(* PLC project marvel_thermovac, Institute of Astronomy Onto 0.0.1 *)
(* stored: creationDateTime 2025-01-01T00:00:00.0, modificationDateTime 2025-01-01T00:00:00.0 *)

{attribute 'qualified_only'}
TYPE TempControlStates : (idle := 0, warming_up := 1, active := 2);
END_TYPE

{attribute 'qualified_only'}
TYPE TempControlStatus : (unknown := 0, invalid_model := 1, idle := 2, warming_up := 3, active := 4) BYTE;
END_TYPE

TYPE OuterRoomParts : STRUCT
  {attribute 'TcHmiSymbol.Show'}
  tFloorE : TempMeasurement;  (* Floor sensor East *)
  {attribute 'TcHmiSymbol.Show'}
  tFloorW : TempMeasurement;  (* Floor sensor West *)
  {attribute 'TcHmiSymbol.Show'}
  tTopN : TempMeasurement;  (* Top sensor North *)
  {attribute 'TcHmiSymbol.Show'}
  tTopS : TempMeasurement;  (* Top sensor South *)
  {attribute 'TcHmiSymbol.Show'}
  ref : RefSensor;  (* Reference 'sensor' for calibration purposes *)
END_STRUCT;
END_TYPE

TYPE InnerRoomParts : STRUCT
  {attribute 'TcHmiSymbol.Show'}
  tAbove : TempMeasurement;  (* 1st temp sensor *)
  {attribute 'TcHmiSymbol.Show'}
  tBelow : TempMeasurement;  (* 2nd temp sensor *)
  {attribute 'TcHmiSymbol.Show'}
  tEast : TempMeasurement;  (* 3rd temp sensor *)
  {attribute 'TcHmiSymbol.Show'}
  tWest : TempMeasurement;  (* 4th temp sensor *)
  {attribute 'TcHmiSymbol.Show'}
  htDucts : Heater;  (* Test heater *)
  {attribute 'TcHmiSymbol.Show'}
  ref : RefSensor;  (* Reference 'sensor' for calibration purposes *)
END_STRUCT;
END_TYPE

TYPE VesselParts : STRUCT
  {attribute 'TcHmiSymbol.Show'}
  tLegNE : TempMeasurement;  (* Leg NE *)
  {attribute 'TcHmiSymbol.Show'}
  tLegNW : TempMeasurement;  (* Leg NW *)
  {attribute 'TcHmiSymbol.Show'}
  tLegSE : TempMeasurement;  (* Leg SE *)
  {attribute 'TcHmiSymbol.Show'}
  tLegSW : TempMeasurement;  (* Leg SW *)
  {attribute 'TcHmiSymbol.Show'}
  tLegTopNE : TempMeasurement;  (* Leg Top NE *)
  {attribute 'TcHmiSymbol.Show'}
  tLegTopNW : TempMeasurement;  (* Leg Top NW *)
  {attribute 'TcHmiSymbol.Show'}
  tLegTopSE : TempMeasurement;  (* Leg Top SE *)
  {attribute 'TcHmiSymbol.Show'}
  tLegTopSW : TempMeasurement;  (* Leg Top SW *)
  {attribute 'TcHmiSymbol.Show'}
  tBotNE : TempMeasurement;  (* Vessel Bottom NE *)
  {attribute 'TcHmiSymbol.Show'}
  tBotNW : TempMeasurement;  (* Vessel Bottom NW *)
  {attribute 'TcHmiSymbol.Show'}
  tBotSE : TempMeasurement;  (* Vessel Bottom SE *)
  {attribute 'TcHmiSymbol.Show'}
  tBotSW : TempMeasurement;  (* Vessel Bottom SW *)
  {attribute 'TcHmiSymbol.Show'}
  tCenter : TempMeasurement;  (* Centre *)
  {attribute 'TcHmiSymbol.Show'}
  tCenterTH10K : TempMeasurement;  (* Centre TH10K *)
  {attribute 'TcHmiSymbol.Show'}
  tSideN : TempMeasurement;  (* Vessel Side N *)
  {attribute 'TcHmiSymbol.Show'}
  tSideS : TempMeasurement;  (* Vessel Side S *)
  {attribute 'TcHmiSymbol.Show'}
  tSideE : TempMeasurement;  (* Vessel Side E *)
  {attribute 'TcHmiSymbol.Show'}
  tSideW : TempMeasurement;  (* Vessel Side W *)
  {attribute 'TcHmiSymbol.Show'}
  tLidN : TempMeasurement;  (* Vessel Lid N *)
  {attribute 'TcHmiSymbol.Show'}
  tLidS : TempMeasurement;  (* Vessel Lid S *)
  {attribute 'TcHmiSymbol.Show'}
  htLegNE : Heater;  (* Heater control for Leg NE *)
  {attribute 'TcHmiSymbol.Show'}
  htLegNW : Heater;  (* Heater control for Leg NW *)
  {attribute 'TcHmiSymbol.Show'}
  htLegSE : Heater;  (* Heater control for Leg SE *)
  {attribute 'TcHmiSymbol.Show'}
  htLegSW : Heater;  (* Heater control for Leg SW *)
  {attribute 'TcHmiSymbol.Show'}
  htLegTopNE : Heater;  (* Heater control for Leg Top NE *)
  {attribute 'TcHmiSymbol.Show'}
  htLegTopNW : Heater;  (* Heater control for Leg Top NW *)
  {attribute 'TcHmiSymbol.Show'}
  htLegTopSE : Heater;  (* Heater control for Leg Top SE *)
  {attribute 'TcHmiSymbol.Show'}
  htLegTopSW : Heater;  (* Heater control for Leg Top SW *)
  {attribute 'TcHmiSymbol.Show'}
  htBotNE : Heater;  (* Heater control for Vessel Bottom NE *)
  {attribute 'TcHmiSymbol.Show'}
  htBotNW : Heater;  (* Heater control for Vessel Bottom NW *)
  {attribute 'TcHmiSymbol.Show'}
  htBotSE : Heater;  (* Heater control for Vessel Bottom SE *)
  {attribute 'TcHmiSymbol.Show'}
  htBotSW : Heater;  (* Heater control for Vessel Bottom SW *)
  {attribute 'TcHmiSymbol.Show'}
  htSideN : Heater;  (* Heater control for Vessel Side NE *)
  {attribute 'TcHmiSymbol.Show'}
  htSideS : Heater;  (* Heater control for Vessel Side NW *)
  {attribute 'TcHmiSymbol.Show'}
  htSideE : Heater;  (* Heater control for Vessel Side SE *)
  {attribute 'TcHmiSymbol.Show'}
  htSideW : Heater;  (* Heater control for Vessel Side SW *)
  {attribute 'TcHmiSymbol.Show'}
  htLidN : Heater;  (* Heater control for Vessel Lid N *)
  {attribute 'TcHmiSymbol.Show'}
  htLidS : Heater;  (* Heater control for Vessel Lid S *)
  {attribute 'TcHmiSymbol.Show'}
  ref : RefSensor;  (* Reference 'sensor' for calibration purposes *)
END_STRUCT;
END_TYPE

TYPE ShieldParts : STRUCT
  {attribute 'TcHmiSymbol.Show'}
  tTopNE : TempMeasurement;  (* Shield top NE *)
  {attribute 'TcHmiSymbol.Show'}
  tTopNW : TempMeasurement;  (* Shield top NW *)
  {attribute 'TcHmiSymbol.Show'}
  tTopSE : TempMeasurement;  (* Shield top SE *)
  {attribute 'TcHmiSymbol.Show'}
  tTopSW : TempMeasurement;  (* Shield top SW *)
  {attribute 'TcHmiSymbol.Show'}
  tSideN : TempMeasurement;  (* Shield side N *)
  {attribute 'TcHmiSymbol.Show'}
  tSideS : TempMeasurement;  (* Shield side S *)
  {attribute 'TcHmiSymbol.Show'}
  tSideNE : TempMeasurement;  (* Shield side NE *)
  {attribute 'TcHmiSymbol.Show'}
  tSideSE : TempMeasurement;  (* Shield side SE *)
  {attribute 'TcHmiSymbol.Show'}
  tSideNW : TempMeasurement;  (* Shield side NW *)
  {attribute 'TcHmiSymbol.Show'}
  tSideSW : TempMeasurement;  (* Shield side SW *)
  {attribute 'TcHmiSymbol.Show'}
  tBotNE : TempMeasurement;  (* Shield bottom NE *)
  {attribute 'TcHmiSymbol.Show'}
  tBotNW : TempMeasurement;  (* Shield bottom NW *)
  {attribute 'TcHmiSymbol.Show'}
  tBotS : TempMeasurement;  (* Shield bottom S *)
  {attribute 'TcHmiSymbol.Show'}
  tCentre : TempMeasurement;  (* Shield centre *)
  {attribute 'TcHmiSymbol.Show'}
  tCentreTh10k : TempMeasurement;  (* Shield centre TH10k *)
  {attribute 'TcHmiSymbol.Show'}
  htTopNE : Heater;  (* Heater control for shield top NE *)
  {attribute 'TcHmiSymbol.Show'}
  htTopNW : Heater;  (* Heater control for shield top NW *)
  {attribute 'TcHmiSymbol.Show'}
  htTopSE : Heater;  (* Heater control for shield top SE *)
  {attribute 'TcHmiSymbol.Show'}
  htTopSW : Heater;  (* Heater control for shield top SW *)
  {attribute 'TcHmiSymbol.Show'}
  htSideN : Heater;  (* Heater control for shield side N *)
  {attribute 'TcHmiSymbol.Show'}
  htSideS : Heater;  (* Heater control for shield side S *)
  {attribute 'TcHmiSymbol.Show'}
  htSideNE : Heater;  (* Heater control for shield side NE *)
  {attribute 'TcHmiSymbol.Show'}
  htSideSE : Heater;  (* Heater control for shield side SE *)
  {attribute 'TcHmiSymbol.Show'}
  htSideNW : Heater;  (* Heater control for shield side NW *)
  {attribute 'TcHmiSymbol.Show'}
  htSideSW : Heater;  (* Heater control for shield side SW *)
  {attribute 'TcHmiSymbol.Show'}
  htBotNE : Heater;  (* Heater control for shield bottom NE *)
  {attribute 'TcHmiSymbol.Show'}
  htBotNW : Heater;  (* Heater control for shield bottom NW *)
  {attribute 'TcHmiSymbol.Show'}
  htBotS : Heater;  (* Heater control for shield bottom S *)
  {attribute 'TcHmiSymbol.Show'}
  htCentre : Heater;  (* Heater control for shield centre *)
  {attribute 'TcHmiSymbol.Show'}
  ref : RefSensor;  (* Reference 'sensor' for calibration purposes *)
END_STRUCT;
END_TYPE

TYPE BenchParts : STRUCT
  {attribute 'TcHmiSymbol.Show'}
  tCentre : TempMeasurement;  (* Bench centre *)
  {attribute 'TcHmiSymbol.Show'}
  tCentreTH10k : TempMeasurement;  (* Bench centre TH10k *)
  {attribute 'TcHmiSymbol.Show'}
  tCollBench : TempMeasurement;  (* Collimator bench *)
  {attribute 'TcHmiSymbol.Show'}
  tEchelleCryo : TempMeasurement;  (* Echelle cryo *)
  {attribute 'TcHmiSymbol.Show'}
  tCamCryo : TempMeasurement;  (* Camera cryo *)
  {attribute 'TcHmiSymbol.Show'}
  tColl : TempMeasurement;  (* Collimator *)
  {attribute 'TcHmiSymbol.Show'}
  tPrism : TempMeasurement;  (* Prism *)
  {attribute 'TcHmiSymbol.Show'}
  tEchelle : TempMeasurement;  (* Echelle *)
  {attribute 'TcHmiSymbol.Show'}
  tCam : TempMeasurement;  (* Camera *)
  {attribute 'TcHmiSymbol.Show'}
  tInOptics : TempMeasurement;  (* In-optics *)
  {attribute 'TcHmiSymbol.Show'}
  htCollBench : Heater;  (* Heater control for collimator bench *)
  {attribute 'TcHmiSymbol.Show'}
  htEchelleCryo : Heater;  (* Heater control for echelle cryo *)
  {attribute 'TcHmiSymbol.Show'}
  htCamCryo : Heater;  (* Heater control for camera cryo *)
  {attribute 'TcHmiSymbol.Show'}
  htEchellePrism : Heater;  (* Heater control for echelle/prism *)
  {attribute 'TcHmiSymbol.Show'}
  ref : RefSensor;  (* Reference 'sensor' for calibration purposes *)
END_STRUCT;
END_TYPE

TYPE CryoParts : STRUCT
  {attribute 'TcHmiSymbol.Show'}
  tRearOut : TempMeasurement;  (* Cryo rear outside *)
  {attribute 'TcHmiSymbol.Show'}
  tRearIn : TempMeasurement;  (* Cryo rear inside *)
  {attribute 'TcHmiSymbol.Show'}
  tFront : TempMeasurement;  (* Cryo front *)
  {attribute 'TcHmiSymbol.Show'}
  htRearOut : Heater;  (* Heater control for cryo rear outside *)
  {attribute 'TcHmiSymbol.Show'}
  htRearIn : Heater;  (* Heater control for cryo rear inside *)
  {attribute 'TcHmiSymbol.Show'}
  htRearFront : Heater;  (* Heater control for cryo front *)
  {attribute 'TcHmiSymbol.Show'}
  ref : RefSensor;  (* Reference 'sensor' for calibration purposes *)
END_STRUCT;
END_TYPE

TYPE ThermoParts : STRUCT
  {attribute 'TcHmiSymbol.Show'}
  outerRoom : OuterRoom;  (* State machine for the outer room temperature control *)
  {attribute 'TcHmiSymbol.Show'}
  innerRoom : InnerRoom;  (* State machine for the inner room temperature control *)
  {attribute 'TcHmiSymbol.Show'}
  vessel : Vessel;  (* State machine for the vessel temperature control *)
  {attribute 'TcHmiSymbol.Show'}
  shield : Shield;  (* State machine for the shield temperature control *)
  {attribute 'TcHmiSymbol.Show'}
  bench : Bench;  (* State machine for the bench temperature control *)
  {attribute 'TcHmiSymbol.Show'}
  cryo : Cryo;  (* State machine for the cryo temperature control *)
END_STRUCT;
END_TYPE

TYPE ThermoVacParts : STRUCT
  {attribute 'TcHmiSymbol.Show'}
  thermo : Thermo;  (* statemachine of the thermal control system *)
  {attribute 'TcHmiSymbol.Show'}
  vac : Vac;  (* statemachine of the vac control system *)
  {attribute 'TcHmiSymbol.Show'}
  configManager : ConfigManager;  (* The config manager (to load/save/activate configuration data) *)
END_STRUCT;
END_TYPE

TYPE TempMeasurementProcesses : STRUCT
  {attribute 'TcHmiSymbol.Show'}
  initialize : Process;  (* Initialize measurement *)
  {attribute 'TcHmiSymbol.Show'}
  clearPtp : Process;  (* Clear PTP values *)
END_STRUCT;
END_TYPE

TYPE HeaterProcesses : STRUCT
  {attribute 'TcHmiSymbol.Show'}
  initialize : Process;  (* Initialize the heater control *)
  {attribute 'TcHmiSymbol.Show'}
  reset : Process;  (* Reset the heater *)
  {attribute 'TcHmiSymbol.Show'}
  force : ForceHeater;  (* Force a certain power output to the heater *)
END_STRUCT;
END_TYPE

TYPE OuterRoomProcesses : STRUCT
  {attribute 'TcHmiSymbol.Show'}
  initialize : Process;  (* Start initializing *)
  {attribute 'TcHmiSymbol.Show'}
  start : Process;  (* Start warming up *)
  {attribute 'TcHmiSymbol.Show'}
  stop : Process;  (* Stop heating *)
  {attribute 'TcHmiSymbol.Show'}
  reset : Process;  (* Reset complete *)
  {attribute 'TcHmiSymbol.Show'}
  clearPtp : Process;  (* Clear the ptp values *)
  {attribute 'TcHmiSymbol.Show'}
  lock : Process;  (* Lock the outerroom control *)
  {attribute 'TcHmiSymbol.Show'}
  unlock : Process;  (* Unlock the outerroom control *)
END_STRUCT;
END_TYPE

TYPE InnerRoomProcesses : STRUCT
  {attribute 'TcHmiSymbol.Show'}
  initialize : Process;  (* Start initializing *)
  {attribute 'TcHmiSymbol.Show'}
  start : Process;  (* Start warming up *)
  {attribute 'TcHmiSymbol.Show'}
  stop : Process;  (* Stop heating *)
  {attribute 'TcHmiSymbol.Show'}
  reset : Process;  (* Reset complete *)
  {attribute 'TcHmiSymbol.Show'}
  clearPtp : Process;  (* Clear the ptp values *)
  {attribute 'TcHmiSymbol.Show'}
  lock : Process;  (* Lock the vessel control (e.g. when the vessel is opened) *)
  {attribute 'TcHmiSymbol.Show'}
  unlock : Process;  (* Unlock the vessel control (e.g. when the vessel is closed) *)
END_STRUCT;
END_TYPE

TYPE VesselProcesses : STRUCT
  {attribute 'TcHmiSymbol.Show'}
  initialize : Process;  (* Start initializing *)
  {attribute 'TcHmiSymbol.Show'}
  start : Process;  (* Start warming up *)
  {attribute 'TcHmiSymbol.Show'}
  stop : Process;  (* Stop heating *)
  {attribute 'TcHmiSymbol.Show'}
  reset : Process;  (* Reset complete *)
  {attribute 'TcHmiSymbol.Show'}
  clearPtp : Process;  (* Clear the ptp values *)
  {attribute 'TcHmiSymbol.Show'}
  lock : Process;  (* Lock the vessel control (e.g. when the vessel is opened) *)
  {attribute 'TcHmiSymbol.Show'}
  unlock : Process;  (* Unlock the vessel control (e.g. when the vessel is closed) *)
END_STRUCT;
END_TYPE

TYPE ShieldProcesses : STRUCT
  {attribute 'TcHmiSymbol.Show'}
  initialize : Process;  (* Start initializing *)
  {attribute 'TcHmiSymbol.Show'}
  start : Process;  (* Start warming up *)
  {attribute 'TcHmiSymbol.Show'}
  stop : Process;  (* Stop heating *)
  {attribute 'TcHmiSymbol.Show'}
  reset : Process;  (* Reset complete *)
  {attribute 'TcHmiSymbol.Show'}
  clearPtp : Process;  (* Clear the ptp values *)
  {attribute 'TcHmiSymbol.Show'}
  lock : Process;  (* Lock the shield control (e.g. when the shield is opened) *)
  {attribute 'TcHmiSymbol.Show'}
  unlock : Process;  (* Unlock the shield control (e.g. when the shield is closed) *)
END_STRUCT;
END_TYPE

TYPE BenchProcesses : STRUCT
  {attribute 'TcHmiSymbol.Show'}
  initialize : Process;  (* Start initializing *)
  {attribute 'TcHmiSymbol.Show'}
  start : Process;  (* Start warming up *)
  {attribute 'TcHmiSymbol.Show'}
  stop : Process;  (* Stop heating *)
  {attribute 'TcHmiSymbol.Show'}
  reset : Process;  (* Reset complete *)
  {attribute 'TcHmiSymbol.Show'}
  clearPtp : Process;  (* Clear the ptp values *)
  {attribute 'TcHmiSymbol.Show'}
  lock : Process;  (* Lock the bench control *)
  {attribute 'TcHmiSymbol.Show'}
  unlock : Process;  (* Unlock the bench control *)
END_STRUCT;
END_TYPE

TYPE CryoProcesses : STRUCT
  {attribute 'TcHmiSymbol.Show'}
  initialize : Process;  (* Start initializing *)
  {attribute 'TcHmiSymbol.Show'}
  start : Process;  (* Start warming up *)
  {attribute 'TcHmiSymbol.Show'}
  stop : Process;  (* Stop heating *)
  {attribute 'TcHmiSymbol.Show'}
  reset : Process;  (* Reset complete *)
  {attribute 'TcHmiSymbol.Show'}
  clearPtp : Process;  (* Clear the ptp values *)
  {attribute 'TcHmiSymbol.Show'}
  lock : Process;  (* Lock the cryo control *)
  {attribute 'TcHmiSymbol.Show'}
  unlock : Process;  (* Unlock the cryo control *)
END_STRUCT;
END_TYPE

TYPE ThermoProcesses : STRUCT
  {attribute 'TcHmiSymbol.Show'}
  initialize : Process;  (* Start initializing *)
  {attribute 'TcHmiSymbol.Show'}
  start : Process;  (* Start warming up *)
  {attribute 'TcHmiSymbol.Show'}
  stop : Process;  (* Stop heating *)
  {attribute 'TcHmiSymbol.Show'}
  clearPtp : Process;  (* Clear the ptp values *)
  {attribute 'TcHmiSymbol.Show'}
  reset : Process;  (* Reset complete *)
  {attribute 'TcHmiSymbol.Show'}
  lock : Process;  (* Lock the vessel control (e.g. when the vessel is opened) *)
  {attribute 'TcHmiSymbol.Show'}
  unlock : Process;  (* Unlock the vessel control (e.g. when the vessel is closed) *)
END_STRUCT;
END_TYPE

TYPE VacProcesses : STRUCT
  {attribute 'TcHmiSymbol.Show'}
  initialize : Process;  (* Start initializing *)
  {attribute 'TcHmiSymbol.Show'}
  reset : Process;  (* Reset complete *)
  {attribute 'TcHmiSymbol.Show'}
  lock : Process;  (* Lock the vessel control (e.g. when the vessel is opened) *)
  {attribute 'TcHmiSymbol.Show'}
  unlock : Process;  (* Unlock the vessel control (e.g. when the vessel is closed) *)
END_STRUCT;
END_TYPE

TYPE ThermoVacProcesses : STRUCT
  {attribute 'TcHmiSymbol.Show'}
  initialize : Process;  (* Start initializing *)
  {attribute 'TcHmiSymbol.Show'}
  reset : Process;  (* Reset complete *)
  {attribute 'TcHmiSymbol.Show'}
  lock : Process;  (* Lock the vessel control (e.g. when the vessel is opened) *)
  {attribute 'TcHmiSymbol.Show'}
  unlock : Process;  (* Unlock the vessel control (e.g. when the vessel is closed) *)
END_STRUCT;
END_TYPE

TYPE TempMeasurementStatuses : STRUCT
  {attribute 'OPC.UA.DA' := '1'}
  {attribute 'OPC.UA.DA.Access' := '1'}
  {attribute 'TcHmiSymbol.Show'}
  init : InitializationStatus;
  {attribute 'OPC.UA.DA' := '1'}
  {attribute 'OPC.UA.DA.Access' := '1'}
  {attribute 'TcHmiSymbol.Show'}
  enabled : EnabledStatus;  (* Is the measurement enabled? *)
  {attribute 'OPC.UA.DA' := '1'}
  {attribute 'OPC.UA.DA.Access' := '1'}
  {attribute 'TcHmiSymbol.Show'}
  health : HealthStatus;  (* Is the measurement OK? *)
  {attribute 'OPC.UA.DA' := '1'}
  {attribute 'OPC.UA.DA.Access' := '1'}
  {attribute 'TcHmiSymbol.Show'}
  alarm : HiHiLoLoAlarmStatus;  (* Alarm status *)
END_STRUCT;
END_TYPE

TYPE HeaterStatuses : STRUCT
  {attribute 'OPC.UA.DA' := '1'}
  {attribute 'OPC.UA.DA.Access' := '1'}
  {attribute 'TcHmiSymbol.Show'}
  init : InitializationStatus;
  {attribute 'OPC.UA.DA' := '1'}
  {attribute 'OPC.UA.DA.Access' := '1'}
  {attribute 'TcHmiSymbol.Show'}
  enabled : EnabledStatus;  (* Is the heater enabled? *)
  {attribute 'OPC.UA.DA' := '1'}
  {attribute 'OPC.UA.DA.Access' := '1'}
  {attribute 'TcHmiSymbol.Show'}
  health : HealthStatus;  (* Is the heater healthy? *)
  {attribute 'OPC.UA.DA' := '1'}
  {attribute 'OPC.UA.DA.Access' := '1'}
  {attribute 'TcHmiSymbol.Show'}
  alarm : HiHiLoLoAlarmStatus;  (* Alarm status *)
END_STRUCT;
END_TYPE

TYPE OuterRoomStatuses : STRUCT
  {attribute 'OPC.UA.DA' := '1'}
  {attribute 'OPC.UA.DA.Access' := '1'}
  {attribute 'TcHmiSymbol.Show'}
  init : InitializationStatus;
  {attribute 'OPC.UA.DA' := '1'}
  {attribute 'OPC.UA.DA.Access' := '1'}
  {attribute 'TcHmiSymbol.Show'}
  enabled : EnabledStatus;  (* Is the outer room enabled? *)
  {attribute 'OPC.UA.DA' := '1'}
  {attribute 'OPC.UA.DA.Access' := '1'}
  {attribute 'TcHmiSymbol.Show'}
  health : HealthStatus;  (* Is the outer room healthy? *)
  {attribute 'OPC.UA.DA' := '1'}
  {attribute 'OPC.UA.DA.Access' := '1'}
  {attribute 'TcHmiSymbol.Show'}
  control : TempControlStatus;  (* Actual state of the outer room *)
  {attribute 'OPC.UA.DA' := '1'}
  {attribute 'OPC.UA.DA.Access' := '1'}
  {attribute 'TcHmiSymbol.Show'}
  busy : BusyStatus;  (* Is the outer room busy with a procedure? *)
END_STRUCT;
END_TYPE

TYPE InnerRoomStatuses : STRUCT
  {attribute 'OPC.UA.DA' := '1'}
  {attribute 'OPC.UA.DA.Access' := '1'}
  {attribute 'TcHmiSymbol.Show'}
  init : InitializationStatus;
  {attribute 'OPC.UA.DA' := '1'}
  {attribute 'OPC.UA.DA.Access' := '1'}
  {attribute 'TcHmiSymbol.Show'}
  enabled : EnabledStatus;  (* Is the inner room enabled? *)
  {attribute 'OPC.UA.DA' := '1'}
  {attribute 'OPC.UA.DA.Access' := '1'}
  {attribute 'TcHmiSymbol.Show'}
  health : HealthStatus;  (* Is the vessel healthy? *)
  {attribute 'OPC.UA.DA' := '1'}
  {attribute 'OPC.UA.DA.Access' := '1'}
  {attribute 'TcHmiSymbol.Show'}
  control : TempControlStatus;  (* Actual state of the vessel *)
  {attribute 'OPC.UA.DA' := '1'}
  {attribute 'OPC.UA.DA.Access' := '1'}
  {attribute 'TcHmiSymbol.Show'}
  busy : BusyStatus;  (* Is the vessel busy with a procedure? *)
END_STRUCT;
END_TYPE

TYPE VesselStatuses : STRUCT
  {attribute 'OPC.UA.DA' := '1'}
  {attribute 'OPC.UA.DA.Access' := '1'}
  {attribute 'TcHmiSymbol.Show'}
  init : InitializationStatus;
  {attribute 'OPC.UA.DA' := '1'}
  {attribute 'OPC.UA.DA.Access' := '1'}
  {attribute 'TcHmiSymbol.Show'}
  enabled : EnabledStatus;  (* Is the vessel enabled? *)
  {attribute 'OPC.UA.DA' := '1'}
  {attribute 'OPC.UA.DA.Access' := '1'}
  {attribute 'TcHmiSymbol.Show'}
  health : HealthStatus;  (* Is the vessel healthy? *)
  {attribute 'OPC.UA.DA' := '1'}
  {attribute 'OPC.UA.DA.Access' := '1'}
  {attribute 'TcHmiSymbol.Show'}
  control : TempControlStatus;  (* Actual state of the vessel *)
  {attribute 'OPC.UA.DA' := '1'}
  {attribute 'OPC.UA.DA.Access' := '1'}
  {attribute 'TcHmiSymbol.Show'}
  busy : BusyStatus;  (* Is the vessel busy with a procedure? *)
END_STRUCT;
END_TYPE

TYPE ShieldStatuses : STRUCT
  {attribute 'OPC.UA.DA' := '1'}
  {attribute 'OPC.UA.DA.Access' := '1'}
  {attribute 'TcHmiSymbol.Show'}
  init : InitializationStatus;
  {attribute 'OPC.UA.DA' := '1'}
  {attribute 'OPC.UA.DA.Access' := '1'}
  {attribute 'TcHmiSymbol.Show'}
  enabled : EnabledStatus;  (* Is the shield enabled? *)
  {attribute 'OPC.UA.DA' := '1'}
  {attribute 'OPC.UA.DA.Access' := '1'}
  {attribute 'TcHmiSymbol.Show'}
  health : HealthStatus;  (* Is the shield healthy? *)
  {attribute 'OPC.UA.DA' := '1'}
  {attribute 'OPC.UA.DA.Access' := '1'}
  {attribute 'TcHmiSymbol.Show'}
  control : TempControlStatus;  (* Actual state of the shield *)
  {attribute 'OPC.UA.DA' := '1'}
  {attribute 'OPC.UA.DA.Access' := '1'}
  {attribute 'TcHmiSymbol.Show'}
  busy : BusyStatus;  (* Is the shield busy with a procedure? *)
END_STRUCT;
END_TYPE

TYPE BenchStatuses : STRUCT
  {attribute 'OPC.UA.DA' := '1'}
  {attribute 'OPC.UA.DA.Access' := '1'}
  {attribute 'TcHmiSymbol.Show'}
  init : InitializationStatus;
  {attribute 'OPC.UA.DA' := '1'}
  {attribute 'OPC.UA.DA.Access' := '1'}
  {attribute 'TcHmiSymbol.Show'}
  enabled : EnabledStatus;  (* Is the bench enabled? *)
  {attribute 'OPC.UA.DA' := '1'}
  {attribute 'OPC.UA.DA.Access' := '1'}
  {attribute 'TcHmiSymbol.Show'}
  health : HealthStatus;  (* Is the bench healthy? *)
  {attribute 'OPC.UA.DA' := '1'}
  {attribute 'OPC.UA.DA.Access' := '1'}
  {attribute 'TcHmiSymbol.Show'}
  control : TempControlStatus;  (* Actual state of the bench *)
  {attribute 'OPC.UA.DA' := '1'}
  {attribute 'OPC.UA.DA.Access' := '1'}
  {attribute 'TcHmiSymbol.Show'}
  busy : BusyStatus;  (* Is the bench busy with a procedure? *)
END_STRUCT;
END_TYPE

TYPE CryoStatuses : STRUCT
  {attribute 'OPC.UA.DA' := '1'}
  {attribute 'OPC.UA.DA.Access' := '1'}
  {attribute 'TcHmiSymbol.Show'}
  init : InitializationStatus;
  {attribute 'OPC.UA.DA' := '1'}
  {attribute 'OPC.UA.DA.Access' := '1'}
  {attribute 'TcHmiSymbol.Show'}
  enabled : EnabledStatus;  (* Is the cryo enabled? *)
  {attribute 'OPC.UA.DA' := '1'}
  {attribute 'OPC.UA.DA.Access' := '1'}
  {attribute 'TcHmiSymbol.Show'}
  health : HealthStatus;  (* Is the cryo healthy? *)
  {attribute 'OPC.UA.DA' := '1'}
  {attribute 'OPC.UA.DA.Access' := '1'}
  {attribute 'TcHmiSymbol.Show'}
  control : TempControlStatus;  (* Actual state of the cryo *)
  {attribute 'OPC.UA.DA' := '1'}
  {attribute 'OPC.UA.DA.Access' := '1'}
  {attribute 'TcHmiSymbol.Show'}
  busy : BusyStatus;  (* Is the cryo busy with a procedure? *)
END_STRUCT;
END_TYPE

TYPE ThermoStatuses : STRUCT
  {attribute 'OPC.UA.DA' := '1'}
  {attribute 'OPC.UA.DA.Access' := '1'}
  {attribute 'TcHmiSymbol.Show'}
  enabled : EnabledStatus;  (* Is the thermo control system enabled? *)
  {attribute 'OPC.UA.DA' := '1'}
  {attribute 'OPC.UA.DA.Access' := '1'}
  {attribute 'TcHmiSymbol.Show'}
  init : InitializationStatus;
  {attribute 'OPC.UA.DA' := '1'}
  {attribute 'OPC.UA.DA.Access' := '1'}
  {attribute 'TcHmiSymbol.Show'}
  health : HealthStatus;  (* Is the healthy? *)
  {attribute 'OPC.UA.DA' := '1'}
  {attribute 'OPC.UA.DA.Access' := '1'}
  {attribute 'TcHmiSymbol.Show'}
  busy : BusyStatus;  (* Is the vessel busy with a procedure? *)
  {attribute 'OPC.UA.DA' := '1'}
  {attribute 'OPC.UA.DA.Access' := '1'}
  {attribute 'TcHmiSymbol.Show'}
  control : TempControlStatus;  (* control state of the thermo control system *)
  {attribute 'OPC.UA.DA' := '1'}
  {attribute 'OPC.UA.DA.Access' := '1'}
  {attribute 'TcHmiSymbol.Show'}
  roomsStatHealth : HealthStatus;  (* Summerization of health states rooms, used for hmi *)
  {attribute 'OPC.UA.DA' := '1'}
  {attribute 'OPC.UA.DA.Access' := '1'}
  {attribute 'TcHmiSymbol.Show'}
  roomsStatBusy : BusyStatus;  (* Summerization of busy states rooms, used for hmi *)
END_STRUCT;
END_TYPE

TYPE VacStatuses : STRUCT
  {attribute 'OPC.UA.DA' := '1'}
  {attribute 'OPC.UA.DA.Access' := '1'}
  {attribute 'TcHmiSymbol.Show'}
  enabled : EnabledStatus;  (* Is the vac system enabled? *)
  {attribute 'OPC.UA.DA' := '1'}
  {attribute 'OPC.UA.DA.Access' := '1'}
  {attribute 'TcHmiSymbol.Show'}
  init : InitializationStatus;
  {attribute 'OPC.UA.DA' := '1'}
  {attribute 'OPC.UA.DA.Access' := '1'}
  {attribute 'TcHmiSymbol.Show'}
  health : HealthStatus;  (* Is the vessel healthy? *)
  {attribute 'OPC.UA.DA' := '1'}
  {attribute 'OPC.UA.DA.Access' := '1'}
  {attribute 'TcHmiSymbol.Show'}
  busy : BusyStatus;  (* Is the vessel busy with a procedure? *)
END_STRUCT;
END_TYPE

TYPE ThermoVacStatuses : STRUCT
  {attribute 'OPC.UA.DA' := '1'}
  {attribute 'OPC.UA.DA.Access' := '1'}
  {attribute 'TcHmiSymbol.Show'}
  init : InitializationStatus;
  {attribute 'OPC.UA.DA' := '1'}
  {attribute 'OPC.UA.DA.Access' := '1'}
  {attribute 'TcHmiSymbol.Show'}
  health : HealthStatus;  (* Is the vessel healthy? *)
  {attribute 'OPC.UA.DA' := '1'}
  {attribute 'OPC.UA.DA.Access' := '1'}
  {attribute 'TcHmiSymbol.Show'}
  busy : BusyStatus;  (* Is the vessel busy with a procedure? *)
END_STRUCT;
END_TYPE

TYPE HeaterConfig : STRUCT
  {attribute 'TcHmiSymbol.Show'}
  enabled : BOOL := TRUE;  (* True if the heater is enabled *)
  {attribute 'TcHmiSymbol.Show'}
  maxPower : LREAL := 100.0;  (* Maximum power of the heater *)
  {attribute 'TcHmiSymbol.Show'}
  Kp : LREAL;  (* proportional gain *)
  {attribute 'TcHmiSymbol.Show'}
  Tn : LREAL;  (* integral gain (in seconds) *)
  {attribute 'TcHmiSymbol.Show'}
  Tv : LREAL;  (* derivative gain D-T1 (in seconds) *)
  {attribute 'TcHmiSymbol.Show'}
  Td : LREAL;  (* derivative damping time D-T1 (in seconds) *)
END_STRUCT;
END_TYPE

TYPE MeasurementConfig2 : STRUCT
  {attribute 'TcHmiSymbol.Show'}
  enabled : BOOL := TRUE;  (* Is the quantity being measured? (Can be false e.g. if the sensor is deliberately not connected (yet).) *)
  {attribute 'TcHmiSymbol.Show'}
  gain : LREAL := 1.0;  (* Gain to be applied to the measured value (default: 1 = no gain) *)
  {attribute 'TcHmiSymbol.Show'}
  offset : LREAL;  (* Offset to be added to the measured value (default: 0 = no offset) *)
END_STRUCT;
END_TYPE

TYPE SimulationConfig : STRUCT
  {attribute 'TcHmiSymbol.Show'}
  ambient : LREAL;  (* starting temp of sensors *)
  {attribute 'TcHmiSymbol.Show'}
  heating : LREAL;  (* heating gain/factor (0-1) *)
  {attribute 'TcHmiSymbol.Show'}
  cooling : LREAL;  (* cooling factor (0-1) *)
  {attribute 'TcHmiSymbol.Show'}
  noise : LREAL;  (* factor (0-1) multiplied with random number (0-1) to create noise in the simulated temperature *)
END_STRUCT;
END_TYPE

TYPE SharedHeaterConfig : STRUCT
  {attribute 'TcHmiSymbol.Show'}
  simulation : SimulationConfig;
  {attribute 'TcHmiSymbol.Show'}
  hihilolo : HiHiLoLoAlarmConfig;  (* Alarm config for the heater's deviation from setpoint *)
  {attribute 'TcHmiSymbol.Show'}
  pwmPeriod : UINT := 1000;  (* period of the pwm signlas in ms *)
  {attribute 'TcHmiSymbol.Show'}
  pwmInstantUpdate : BOOL;  (* True if the PWM signal is updated instantly when the power changes *)
  {attribute 'TcHmiSymbol.Show'}
  maxPower : LREAL := 100.0;  (* Maximum total power of all heaters in percentage *)
  {attribute 'TcHmiSymbol.Show'}
  pidCycleTime : UINT := 100;  (* cycle time of the heater control loop in ms *)
  {attribute 'TcHmiSymbol.Show'}
  arwOnlyIpart : BOOL := TRUE;  (* True if the anti reset windup only applies to the integral part of the PID controller *)
END_STRUCT;
END_TYPE

TYPE SharedMeasurementConfig : STRUCT
  {attribute 'TcHmiSymbol.Show'}
  alarms : HiHiLoLoAlarmConfig;  (* Alarm config for the temperature sensors *)
  {attribute 'TcHmiSymbol.Show'}
  cycleTime : UINT := 100;  (* time in ms between temp measurements *)
  {attribute 'TcHmiSymbol.Show'}
  nrOfSamples : UINT := 50;  (* number of samples of the moving average *)
END_STRUCT;
END_TYPE

TYPE OuterRoomSharedConfig : STRUCT
  {attribute 'TcHmiSymbol.Show'}
  sensors : SharedMeasurementConfig;  (* Shared config for the temperature sensors *)
END_STRUCT;
END_TYPE

TYPE InnerRoomSharedConfig : STRUCT
  {attribute 'TcHmiSymbol.Show'}
  sensors : SharedMeasurementConfig;  (* Shared config for the temperature sensors *)
  {attribute 'TcHmiSymbol.Show'}
  heaters : SharedHeaterConfig;  (* Shared config for the heaters *)
END_STRUCT;
END_TYPE

TYPE VesselSharedConfig : STRUCT
  {attribute 'TcHmiSymbol.Show'}
  sensors : SharedMeasurementConfig;  (* Shared config for the temperature sensors in the vessel *)
  {attribute 'TcHmiSymbol.Show'}
  heaters : SharedHeaterConfig;  (* Shared config for the heaters in the vessel *)
END_STRUCT;
END_TYPE

TYPE ShieldSharedConfig : STRUCT
  {attribute 'TcHmiSymbol.Show'}
  sensors : SharedMeasurementConfig;  (* Shared config for the temperature sensors in the shield *)
  {attribute 'TcHmiSymbol.Show'}
  heaters : SharedHeaterConfig;  (* Shared config for the heaters in the shield *)
END_STRUCT;
END_TYPE

TYPE BenchSharedConfig : STRUCT
  {attribute 'TcHmiSymbol.Show'}
  sensors : SharedMeasurementConfig;  (* Shared config for the temperature sensors in the bench *)
  {attribute 'TcHmiSymbol.Show'}
  heaters : SharedHeaterConfig;  (* Shared config for the heaters in the bench *)
END_STRUCT;
END_TYPE

TYPE CryoSharedConfig : STRUCT
  {attribute 'TcHmiSymbol.Show'}
  sensors : SharedMeasurementConfig;  (* Shared config for the temperature sensors in the cryo *)
  {attribute 'TcHmiSymbol.Show'}
  heaters : SharedHeaterConfig;  (* Shared config for the heaters in the cryo *)
END_STRUCT;
END_TYPE

TYPE ThermoSharedConfig : STRUCT
  {attribute 'TcHmiSymbol.Show'}
  placeHolder : BOOL;  (* placeholder for the shared config of the thermo system, can be extended in the future *)
END_STRUCT;
END_TYPE

TYPE OuterRoomConfig : STRUCT
  {attribute 'TcHmiSymbol.Show'}
  enabled : BOOL := TRUE;  (* True if the outer room is enabled *)
  {attribute 'TcHmiSymbol.Show'}
  shared : OuterRoomSharedConfig;  (* Shared config for the outer room *)
  {attribute 'TcHmiSymbol.Show'}
  tFloorE : MeasurementConfig2;  (* Config for floor sensor East *)
  {attribute 'TcHmiSymbol.Show'}
  tFloorW : MeasurementConfig2;  (* Config for floor sensor West *)
  {attribute 'TcHmiSymbol.Show'}
  tTopN : MeasurementConfig2;  (* Config for top sensor North *)
  {attribute 'TcHmiSymbol.Show'}
  tTopS : MeasurementConfig2;  (* Config for top sensor South *)
END_STRUCT;
END_TYPE

TYPE InnerRoomConfig : STRUCT
  {attribute 'TcHmiSymbol.Show'}
  enabled : BOOL := TRUE;  (* True if the inner room is enabled *)
  {attribute 'TcHmiSymbol.Show'}
  shared : InnerRoomSharedConfig;  (* Config shared by inner room's parts *)
  {attribute 'TcHmiSymbol.Show'}
  isSimulated : BOOL;  (* True if the innerroom temperature control is in simulation mode *)
  {attribute 'TcHmiSymbol.Show'}
  setPointTarget : LREAL;  (* set point temperature in celsius *)
  {attribute 'TcHmiSymbol.Show'}
  rampVPos : LREAL;  (* velocity of temperature change in C/s while ramping up *)
  {attribute 'TcHmiSymbol.Show'}
  rampVNeg : LREAL;  (* velocity of temperature change in C/s while ramping down *)
  {attribute 'TcHmiSymbol.Show'}
  rampStart : LREAL;  (* temperature in celsius at which the ramp starts *)
  {attribute 'TcHmiSymbol.Show'}
  hihiPtp : LREAL;  (* Ptp value at which an alarm is given *)
  {attribute 'TcHmiSymbol.Show'}
  hiPtp : LREAL;  (* Ptp value at which a warning is given *)
  {attribute 'TcHmiSymbol.Show'}
  maxInitTime : LREAL := 120.0;  (* Maximum time in seconds before initialization is failed *)
  {attribute 'TcHmiSymbol.Show'}
  minSenRequired : INT := 4;  (* minimum number of sensors required to stay in operation *)
  {attribute 'TcHmiSymbol.Show'}
  tAbove : MeasurementConfig2;  (* Config for temp sensor above the vessel *)
  {attribute 'TcHmiSymbol.Show'}
  tBelow : MeasurementConfig2;  (* Config for temp sensor below the vessel *)
  {attribute 'TcHmiSymbol.Show'}
  tEast : MeasurementConfig2;  (* Config for temp sensor East of the vessel *)
  {attribute 'TcHmiSymbol.Show'}
  tWest : MeasurementConfig2;  (* Config for temp sensor West of the vessel *)
  {attribute 'TcHmiSymbol.Show'}
  htDucts : HeaterConfig;  (* Config for test heater *)
END_STRUCT;
END_TYPE

TYPE VesselConfig : STRUCT
  {attribute 'TcHmiSymbol.Show'}
  enabled : BOOL := TRUE;  (* True if the vessel is enabled *)
  {attribute 'TcHmiSymbol.Show'}
  shared : InnerRoomSharedConfig;  (* Config shared by vessels's parts *)
  {attribute 'TcHmiSymbol.Show'}
  isSimulated : BOOL;  (* True if the vessel temperature control is in simulation mode *)
  {attribute 'TcHmiSymbol.Show'}
  setPointTarget : LREAL;  (* set point temperature in celsius *)
  {attribute 'TcHmiSymbol.Show'}
  rampVPos : LREAL;  (* velocity of temperature change in C/s while ramping up *)
  {attribute 'TcHmiSymbol.Show'}
  rampVNeg : LREAL;  (* velocity of temperature change in C/s while ramping down *)
  {attribute 'TcHmiSymbol.Show'}
  rampStart : LREAL;  (* temperature in celsius at which the ramp starts *)
  {attribute 'TcHmiSymbol.Show'}
  hihiPtp : LREAL;  (* Ptp value at which an alarm is given *)
  {attribute 'TcHmiSymbol.Show'}
  hiPtp : LREAL;  (* Ptp value at which a warning is given *)
  {attribute 'TcHmiSymbol.Show'}
  maxInitTime : LREAL := 120.0;  (* Maximum time in seconds before initialization is failed *)
  {attribute 'TcHmiSymbol.Show'}
  tLegNE : MeasurementConfig2;  (* Config for Leg NE *)
  {attribute 'TcHmiSymbol.Show'}
  tLegNW : MeasurementConfig2;  (* Config for Leg NW *)
  {attribute 'TcHmiSymbol.Show'}
  tLegSE : MeasurementConfig2;  (* Config for Leg SE *)
  {attribute 'TcHmiSymbol.Show'}
  tLegSW : MeasurementConfig2;  (* Config for Leg SW *)
  {attribute 'TcHmiSymbol.Show'}
  tLegTopNE : MeasurementConfig2;  (* Config for Leg Top NE *)
  {attribute 'TcHmiSymbol.Show'}
  tLegTopNW : MeasurementConfig2;  (* Config for Leg Top NW *)
  {attribute 'TcHmiSymbol.Show'}
  tLegTopSE : MeasurementConfig2;  (* Config for Leg Top SE *)
  {attribute 'TcHmiSymbol.Show'}
  tLegTopSW : MeasurementConfig2;  (* Config for Leg Top SW *)
  {attribute 'TcHmiSymbol.Show'}
  tBotNE : MeasurementConfig2;  (* Config for Vessel Bottom NE *)
  {attribute 'TcHmiSymbol.Show'}
  tBotNW : MeasurementConfig2;  (* Config for Vessel Bottom NW *)
  {attribute 'TcHmiSymbol.Show'}
  tBotSE : MeasurementConfig2;  (* Config for Vessel Bottom SE *)
  {attribute 'TcHmiSymbol.Show'}
  tBotSW : MeasurementConfig2;  (* Config for Vessel Bottom SW *)
  {attribute 'TcHmiSymbol.Show'}
  tCenter : MeasurementConfig2;  (* Config for Centre *)
  {attribute 'TcHmiSymbol.Show'}
  tCenterTH10K : MeasurementConfig2;  (* Config for Centre TH10K *)
  {attribute 'TcHmiSymbol.Show'}
  tSideN : MeasurementConfig2;  (* Config for Vessel Side N *)
  {attribute 'TcHmiSymbol.Show'}
  tSideS : MeasurementConfig2;  (* Config for Vessel Side S *)
  {attribute 'TcHmiSymbol.Show'}
  tSideE : MeasurementConfig2;  (* Config for Vessel Side E *)
  {attribute 'TcHmiSymbol.Show'}
  tSideW : MeasurementConfig2;  (* Config for Vessel Side W *)
  {attribute 'TcHmiSymbol.Show'}
  tLidN : MeasurementConfig2;  (* Config for Vessel Lid N *)
  {attribute 'TcHmiSymbol.Show'}
  tLidS : MeasurementConfig2;  (* Config for Vessel Lid S *)
  {attribute 'TcHmiSymbol.Show'}
  htLegNE : HeaterConfig;  (* Config for heater Leg NE *)
  {attribute 'TcHmiSymbol.Show'}
  htLegNW : HeaterConfig;  (* Config for heater Leg NW *)
  {attribute 'TcHmiSymbol.Show'}
  htLegSE : HeaterConfig;  (* Config for heater Leg SE *)
  {attribute 'TcHmiSymbol.Show'}
  htLegSW : HeaterConfig;  (* Config for heater Leg SW *)
  {attribute 'TcHmiSymbol.Show'}
  htLegTopNE : HeaterConfig;  (* Config for heater Leg Top NE *)
  {attribute 'TcHmiSymbol.Show'}
  htLegTopNW : HeaterConfig;  (* Config for heater Leg Top NW *)
  {attribute 'TcHmiSymbol.Show'}
  htLegTopSE : HeaterConfig;  (* Config for heater Leg Top SE *)
  {attribute 'TcHmiSymbol.Show'}
  htLegTopSW : HeaterConfig;  (* Config for heater Leg Top SW *)
  {attribute 'TcHmiSymbol.Show'}
  htBotNE : HeaterConfig;  (* Config for heater Vessel Bottom NE *)
  {attribute 'TcHmiSymbol.Show'}
  htBotNW : HeaterConfig;  (* Config for heater Vessel Bottom NW *)
  {attribute 'TcHmiSymbol.Show'}
  htBotSE : HeaterConfig;  (* Config for heater Vessel Bottom SE *)
  {attribute 'TcHmiSymbol.Show'}
  htBotSW : HeaterConfig;  (* Config for heater Vessel Bottom SW *)
  {attribute 'TcHmiSymbol.Show'}
  htSideN : HeaterConfig;  (* Config for heater Vessel Side NE *)
  {attribute 'TcHmiSymbol.Show'}
  htSideS : HeaterConfig;  (* Config for heater Vessel Side NW *)
  {attribute 'TcHmiSymbol.Show'}
  htSideE : HeaterConfig;  (* Config for heater Vessel Side SE *)
  {attribute 'TcHmiSymbol.Show'}
  htSideW : HeaterConfig;  (* Config for heater Vessel Side SW *)
  {attribute 'TcHmiSymbol.Show'}
  htLidN : HeaterConfig;  (* Config for heater Vessel Lid N *)
  {attribute 'TcHmiSymbol.Show'}
  htLidS : HeaterConfig;  (* Config for heater Vessel Lid S *)
END_STRUCT;
END_TYPE

TYPE ShieldConfig : STRUCT
  {attribute 'TcHmiSymbol.Show'}
  enabled : BOOL := TRUE;  (* True if the shield is enabled *)
  {attribute 'TcHmiSymbol.Show'}
  shared : InnerRoomSharedConfig;  (* Config shared by shield's parts *)
  {attribute 'TcHmiSymbol.Show'}
  isSimulated : BOOL;  (* True if the shield temperature control is in simulation mode *)
  {attribute 'TcHmiSymbol.Show'}
  setPointTarget : LREAL;  (* set point temperature in celsius *)
  {attribute 'TcHmiSymbol.Show'}
  rampVPos : LREAL;  (* velocity of temperature change in C/s while ramping up *)
  {attribute 'TcHmiSymbol.Show'}
  rampVNeg : LREAL;  (* velocity of temperature change in C/s while ramping down *)
  {attribute 'TcHmiSymbol.Show'}
  rampStart : LREAL;  (* temperature in celsius at which the ramp starts *)
  {attribute 'TcHmiSymbol.Show'}
  hihiPtp : LREAL;  (* Ptp value at which an alarm is given *)
  {attribute 'TcHmiSymbol.Show'}
  hiPtp : LREAL;  (* Ptp value at which a warning is given *)
  {attribute 'TcHmiSymbol.Show'}
  maxInitTime : LREAL := 120.0;  (* Maximum time in seconds before initialization is failed *)
  {attribute 'TcHmiSymbol.Show'}
  tTopNE : MeasurementConfig2;  (* Config for shield top NE *)
  {attribute 'TcHmiSymbol.Show'}
  tTopNW : MeasurementConfig2;  (* Config for shield top NW *)
  {attribute 'TcHmiSymbol.Show'}
  tTopSE : MeasurementConfig2;  (* Config for shield top SE *)
  {attribute 'TcHmiSymbol.Show'}
  tTopSW : MeasurementConfig2;  (* Config for shield top SW *)
  {attribute 'TcHmiSymbol.Show'}
  tSideN : MeasurementConfig2;  (* Config for shield side N *)
  {attribute 'TcHmiSymbol.Show'}
  tSideS : MeasurementConfig2;  (* Config for shield side S *)
  {attribute 'TcHmiSymbol.Show'}
  tSideNE : MeasurementConfig2;  (* Config for shield side NE *)
  {attribute 'TcHmiSymbol.Show'}
  tSideSE : MeasurementConfig2;  (* Config for shield side SE *)
  {attribute 'TcHmiSymbol.Show'}
  tSideNW : MeasurementConfig2;  (* Config for shield side NW *)
  {attribute 'TcHmiSymbol.Show'}
  tSideSW : MeasurementConfig2;  (* Config for shield side SW *)
  {attribute 'TcHmiSymbol.Show'}
  tBotNE : MeasurementConfig2;  (* Config for shield bottom NE *)
  {attribute 'TcHmiSymbol.Show'}
  tBotNW : MeasurementConfig2;  (* Config for shield bottom NW *)
  {attribute 'TcHmiSymbol.Show'}
  tBotS : MeasurementConfig2;  (* Config for shield bottom S *)
  {attribute 'TcHmiSymbol.Show'}
  tCentre : MeasurementConfig2;  (* Config for shield centre *)
  {attribute 'TcHmiSymbol.Show'}
  tCentreTh10k : MeasurementConfig2;  (* Config for shield centre TH10k *)
  {attribute 'TcHmiSymbol.Show'}
  htTopNE : HeaterConfig;  (* Config for heater shield top NE *)
  {attribute 'TcHmiSymbol.Show'}
  htTopNW : HeaterConfig;  (* Config for heater shield top NW *)
  {attribute 'TcHmiSymbol.Show'}
  htTopSE : HeaterConfig;  (* Config for heater shield top SE *)
  {attribute 'TcHmiSymbol.Show'}
  htTopSW : HeaterConfig;  (* Config for heater shield top SW *)
  {attribute 'TcHmiSymbol.Show'}
  htSideN : HeaterConfig;  (* Config for heater shield side N *)
  {attribute 'TcHmiSymbol.Show'}
  htSideS : HeaterConfig;  (* Config for heater shield side S *)
  {attribute 'TcHmiSymbol.Show'}
  htSideNE : HeaterConfig;  (* Config for heater shield side NE *)
  {attribute 'TcHmiSymbol.Show'}
  htSideSE : HeaterConfig;  (* Config for heater shield side SE *)
  {attribute 'TcHmiSymbol.Show'}
  htSideNW : HeaterConfig;  (* Config for heater shield side NW *)
  {attribute 'TcHmiSymbol.Show'}
  htSideSW : HeaterConfig;  (* Config for heater shield side SW *)
  {attribute 'TcHmiSymbol.Show'}
  htBotNE : HeaterConfig;  (* Config for heater shield bottom NE *)
  {attribute 'TcHmiSymbol.Show'}
  htBotNW : HeaterConfig;  (* Config for heater shield bottom NW *)
  {attribute 'TcHmiSymbol.Show'}
  htBotS : HeaterConfig;  (* Config for heater shield bottom S *)
  {attribute 'TcHmiSymbol.Show'}
  htCentre : HeaterConfig;  (* Config for heater shield centre *)
END_STRUCT;
END_TYPE

TYPE BenchConfig : STRUCT
  {attribute 'TcHmiSymbol.Show'}
  enabled : BOOL := TRUE;  (* True if bench enabled *)
  {attribute 'TcHmiSymbol.Show'}
  shared : BenchSharedConfig;  (* Bench shared config *)
  {attribute 'TcHmiSymbol.Show'}
  tCentre : MeasurementConfig2;  (* Config for bench centre *)
  {attribute 'TcHmiSymbol.Show'}
  tCentreTH10k : MeasurementConfig2;  (* Bench centre TH10k sensor *)
  {attribute 'TcHmiSymbol.Show'}
  tCollBench : MeasurementConfig2;  (* Config for collimator bench *)
  {attribute 'TcHmiSymbol.Show'}
  tEchelleCryo : MeasurementConfig2;  (* Config for echelle cryo *)
  {attribute 'TcHmiSymbol.Show'}
  tCamCryo : MeasurementConfig2;  (* Config for camera cryo *)
  {attribute 'TcHmiSymbol.Show'}
  tColl : MeasurementConfig2;  (* Config for collimator *)
  {attribute 'TcHmiSymbol.Show'}
  tPrism : MeasurementConfig2;  (* Config for prism *)
  {attribute 'TcHmiSymbol.Show'}
  tEchelle : MeasurementConfig2;  (* Config for echelle *)
  {attribute 'TcHmiSymbol.Show'}
  tCam : MeasurementConfig2;  (* Config for camera *)
  {attribute 'TcHmiSymbol.Show'}
  tInOptics : MeasurementConfig2;  (* Config for in-optics *)
  {attribute 'TcHmiSymbol.Show'}
  htCollBench : HeaterConfig;  (* Config for heater collimator bench *)
  {attribute 'TcHmiSymbol.Show'}
  htEchelleCryo : HeaterConfig;  (* Config for heater echelle cryo *)
  {attribute 'TcHmiSymbol.Show'}
  htCamCryo : HeaterConfig;  (* Config for heater camera cryo *)
  {attribute 'TcHmiSymbol.Show'}
  htEchellePrism : HeaterConfig;  (* Config for heater echelle/prism *)
END_STRUCT;
END_TYPE

TYPE CryoConfig : STRUCT
  {attribute 'TcHmiSymbol.Show'}
  enabled : BOOL := TRUE;  (* True if cryo enabled *)
  {attribute 'TcHmiSymbol.Show'}
  shared : CryoSharedConfig;  (* Cryo shared config *)
  {attribute 'TcHmiSymbol.Show'}
  tRearOut : MeasurementConfig2;  (* Cryo rear outside sensor *)
  {attribute 'TcHmiSymbol.Show'}
  tRearIn : MeasurementConfig2;  (* Cryo rear inside sensor *)
  {attribute 'TcHmiSymbol.Show'}
  tFront : MeasurementConfig2;  (* Cryo front sensor *)
  {attribute 'TcHmiSymbol.Show'}
  htRearOut : HeaterConfig;  (* Heater cryo rear outside *)
  {attribute 'TcHmiSymbol.Show'}
  htRearIn : HeaterConfig;  (* Heater cryo rear inside *)
  {attribute 'TcHmiSymbol.Show'}
  htRearFront : HeaterConfig;  (* Heater cryo front *)
END_STRUCT;
END_TYPE

TYPE ThermoConfig : STRUCT
  {attribute 'TcHmiSymbol.Show'}
  enabled : BOOL := TRUE;  (* True if thermo enabled *)
  {attribute 'TcHmiSymbol.Show'}
  outerRoom : OuterRoomConfig;  (* Config for the outer room *)
  {attribute 'TcHmiSymbol.Show'}
  innerRoom : InnerRoomConfig;  (* Config for the inner room *)
  {attribute 'TcHmiSymbol.Show'}
  vessel : VesselConfig;  (* Config for the vessel *)
  {attribute 'TcHmiSymbol.Show'}
  shield : ShieldConfig;  (* Config for the shield *)
  {attribute 'TcHmiSymbol.Show'}
  bench : BenchConfig;  (* Config for the bench *)
  {attribute 'TcHmiSymbol.Show'}
  cryo : CryoConfig;  (* Config for the cryo *)
  {attribute 'TcHmiSymbol.Show'}
  shared : ThermoSharedConfig;  (* Shared config for the thermo system *)
END_STRUCT;
END_TYPE

TYPE VacConfig : STRUCT
  {attribute 'TcHmiSymbol.Show'}
  enabled : BOOL;  (* True if the vac system is enabled *)
END_STRUCT;
END_TYPE

TYPE ThermoVacConfig : STRUCT
  {attribute 'TcHmiSymbol.Show'}
  thermo : ThermoConfig;  (* Thermo config *)
  {attribute 'TcHmiSymbol.Show'}
  vac : VacConfig;  (* Vacuum config *)
END_STRUCT;
END_TYPE

TYPE ForceHeaterArgs : STRUCT
  {attribute 'TcHmiSymbol.Show'}
  power : REAL;
END_STRUCT;
END_TYPE

TYPE M_SM_RefSensor : STRUCT
  {attribute 'OPC.UA.DA' := '1'}
  {attribute 'OPC.UA.DA.Access' := '1'}
  {attribute 'TcHmiSymbol.Show'}
  actualStatus : STRING;
  {attribute 'OPC.UA.DA' := '1'}
  {attribute 'OPC.UA.DA.Access' := '1'}
  {attribute 'TcHmiSymbol.Show'}
  value : LREAL;
END_STRUCT;
END_TYPE

TYPE M_SM_TempMeasurement : STRUCT
  {attribute 'OPC.UA.DA' := '1'}
  {attribute 'OPC.UA.DA.Access' := '1'}
  {attribute 'TcHmiSymbol.Show'}
  isSimulated : BOOL;
  {attribute 'OPC.UA.DA' := '1'}
  {attribute 'OPC.UA.DA.Access' := '1'}
  {attribute 'TcHmiSymbol.Show'}
  actualStatus : STRING;
  {attribute 'OPC.UA.DA' := '1'}
  {attribute 'OPC.UA.DA.Access' := '1'}
  {attribute 'TcHmiSymbol.Show'}
  value : LREAL;
  {attribute 'OPC.UA.DA' := '1'}
  {attribute 'OPC.UA.DA.Access' := '1'}
  {attribute 'TcHmiSymbol.Show'}
  ptp1 : LREAL;
  {attribute 'OPC.UA.DA' := '1'}
  {attribute 'OPC.UA.DA.Access' := '1'}
  {attribute 'TcHmiSymbol.Show'}
  ptp2 : LREAL;
  {attribute 'OPC.UA.DA' := '1'}
  {attribute 'TcHmiSymbol.Show'}
  stat : TempMeasurementStatuses;
  {attribute 'OPC.UA.DA' := '1'}
  {attribute 'TcHmiSymbol.Show'}
  proc : M_SM_TempMeasurementProcesses;
END_STRUCT;
END_TYPE

TYPE M_SM_Heater : STRUCT
  {attribute 'OPC.UA.DA' := '1'}
  {attribute 'OPC.UA.DA.Access' := '1'}
  {attribute 'TcHmiSymbol.Show'}
  setPoint : LREAL;
  {attribute 'OPC.UA.DA' := '1'}
  {attribute 'OPC.UA.DA.Access' := '1'}
  {attribute 'TcHmiSymbol.Show'}
  temp : LREAL;
  {attribute 'OPC.UA.DA' := '1'}
  {attribute 'OPC.UA.DA.Access' := '1'}
  {attribute 'TcHmiSymbol.Show'}
  isSimulated : BOOL;
  {attribute 'OPC.UA.DA' := '1'}
  {attribute 'OPC.UA.DA.Access' := '1'}
  {attribute 'TcHmiSymbol.Show'}
  actualStatus : STRING;
  {attribute 'OPC.UA.DA' := '1'}
  {attribute 'OPC.UA.DA.Access' := '1'}
  {attribute 'TcHmiSymbol.Show'}
  power : LREAL;
  {attribute 'OPC.UA.DA' := '1'}
  {attribute 'OPC.UA.DA.Access' := '1'}
  {attribute 'TcHmiSymbol.Show'}
  deviation : LREAL;
  {attribute 'OPC.UA.DA' := '1'}
  {attribute 'OPC.UA.DA.Access' := '1'}
  {attribute 'TcHmiSymbol.Show'}
  isForced : BOOL;
  {attribute 'OPC.UA.DA' := '1'}
  {attribute 'OPC.UA.DA.Access' := '1'}
  {attribute 'TcHmiSymbol.Show'}
  simTemp : LREAL;
  {attribute 'OPC.UA.DA' := '1'}
  {attribute 'TcHmiSymbol.Show'}
  stat : HeaterStatuses;
  {attribute 'OPC.UA.DA' := '1'}
  {attribute 'TcHmiSymbol.Show'}
  proc : M_SM_HeaterProcesses;
END_STRUCT;
END_TYPE

TYPE M_SM_OuterRoom : STRUCT
  {attribute 'OPC.UA.DA' := '1'}
  {attribute 'OPC.UA.DA.Access' := '1'}
  {attribute 'TcHmiSymbol.Show'}
  actualStatus : STRING;
  {attribute 'OPC.UA.DA' := '1'}
  {attribute 'TcHmiSymbol.Show'}
  stat : OuterRoomStatuses;
  {attribute 'OPC.UA.DA' := '1'}
  {attribute 'TcHmiSymbol.Show'}
  parts : M_SM_OuterRoomParts;
  {attribute 'OPC.UA.DA' := '1'}
  {attribute 'TcHmiSymbol.Show'}
  proc : M_SM_OuterRoomProcesses;
END_STRUCT;
END_TYPE

TYPE M_SM_InnerRoom : STRUCT
  {attribute 'OPC.UA.DA' := '1'}
  {attribute 'OPC.UA.DA.Access' := '1'}
  {attribute 'TcHmiSymbol.Show'}
  actualStatus : STRING;
  {attribute 'OPC.UA.DA' := '1'}
  {attribute 'OPC.UA.DA.Access' := '1'}
  {attribute 'TcHmiSymbol.Show'}
  setPoint : LREAL;
  {attribute 'OPC.UA.DA' := '1'}
  {attribute 'OPC.UA.DA.Access' := '1'}
  {attribute 'TcHmiSymbol.Show'}
  avgTemp : LREAL;
  {attribute 'OPC.UA.DA' := '1'}
  {attribute 'OPC.UA.DA.Access' := '1'}
  {attribute 'TcHmiSymbol.Show'}
  avgPower : LREAL;
  {attribute 'OPC.UA.DA' := '1'}
  {attribute 'OPC.UA.DA.Access' := '1'}
  {attribute 'TcHmiSymbol.Show'}
  totalPower : LREAL;
  {attribute 'OPC.UA.DA' := '1'}
  {attribute 'OPC.UA.DA.Access' := '1'}
  {attribute 'TcHmiSymbol.Show'}
  ptpAvgTemp : ARRAY[1..5] OF LREAL;
  {attribute 'OPC.UA.DA' := '1'}
  {attribute 'OPC.UA.DA.Access' := '1'}
  {attribute 'TcHmiSymbol.Show'}
  ptpAllTemp : ARRAY[1..5] OF LREAL;
  {attribute 'OPC.UA.DA' := '1'}
  {attribute 'TcHmiSymbol.Show'}
  stat : InnerRoomStatuses;
  {attribute 'OPC.UA.DA' := '1'}
  {attribute 'TcHmiSymbol.Show'}
  parts : M_SM_InnerRoomParts;
  {attribute 'OPC.UA.DA' := '1'}
  {attribute 'TcHmiSymbol.Show'}
  proc : M_SM_InnerRoomProcesses;
END_STRUCT;
END_TYPE

TYPE M_SM_Vessel : STRUCT
  {attribute 'OPC.UA.DA' := '1'}
  {attribute 'OPC.UA.DA.Access' := '1'}
  {attribute 'TcHmiSymbol.Show'}
  tStatBottomOk : BOOL;
  {attribute 'OPC.UA.DA' := '1'}
  {attribute 'OPC.UA.DA.Access' := '1'}
  {attribute 'TcHmiSymbol.Show'}
  tStatLidOk : BOOL;
  {attribute 'OPC.UA.DA' := '1'}
  {attribute 'OPC.UA.DA.Access' := '1'}
  {attribute 'TcHmiSymbol.Show'}
  actualStatus : STRING;
  {attribute 'OPC.UA.DA' := '1'}
  {attribute 'OPC.UA.DA.Access' := '1'}
  {attribute 'TcHmiSymbol.Show'}
  setPoint : LREAL;
  {attribute 'OPC.UA.DA' := '1'}
  {attribute 'OPC.UA.DA.Access' := '1'}
  {attribute 'TcHmiSymbol.Show'}
  avgTemp : LREAL;
  {attribute 'OPC.UA.DA' := '1'}
  {attribute 'OPC.UA.DA.Access' := '1'}
  {attribute 'TcHmiSymbol.Show'}
  avgPower : LREAL;
  {attribute 'OPC.UA.DA' := '1'}
  {attribute 'OPC.UA.DA.Access' := '1'}
  {attribute 'TcHmiSymbol.Show'}
  totalPower : LREAL;
  {attribute 'OPC.UA.DA' := '1'}
  {attribute 'OPC.UA.DA.Access' := '1'}
  {attribute 'TcHmiSymbol.Show'}
  ptpAvgTemp : ARRAY[1..5] OF LREAL;
  {attribute 'OPC.UA.DA' := '1'}
  {attribute 'OPC.UA.DA.Access' := '1'}
  {attribute 'TcHmiSymbol.Show'}
  ptpAllTemp : ARRAY[1..5] OF LREAL;
  {attribute 'OPC.UA.DA' := '1'}
  {attribute 'OPC.UA.DA.Access' := '1'}
  {attribute 'TcHmiSymbol.Show'}
  tStatBottomPwr : BOOL;
  {attribute 'OPC.UA.DA' := '1'}
  {attribute 'OPC.UA.DA.Access' := '1'}
  {attribute 'TcHmiSymbol.Show'}
  tStatLidPwr : BOOL;
  {attribute 'OPC.UA.DA' := '1'}
  {attribute 'TcHmiSymbol.Show'}
  stat : VesselStatuses;
  {attribute 'OPC.UA.DA' := '1'}
  {attribute 'TcHmiSymbol.Show'}
  parts : M_SM_VesselParts;
  {attribute 'OPC.UA.DA' := '1'}
  {attribute 'TcHmiSymbol.Show'}
  proc : M_SM_VesselProcesses;
END_STRUCT;
END_TYPE

TYPE M_SM_Shield : STRUCT
  {attribute 'OPC.UA.DA' := '1'}
  {attribute 'OPC.UA.DA.Access' := '1'}
  {attribute 'TcHmiSymbol.Show'}
  actualStatus : STRING;
  {attribute 'OPC.UA.DA' := '1'}
  {attribute 'OPC.UA.DA.Access' := '1'}
  {attribute 'TcHmiSymbol.Show'}
  setPoint : LREAL;
  {attribute 'OPC.UA.DA' := '1'}
  {attribute 'OPC.UA.DA.Access' := '1'}
  {attribute 'TcHmiSymbol.Show'}
  avgTemp : LREAL;
  {attribute 'OPC.UA.DA' := '1'}
  {attribute 'OPC.UA.DA.Access' := '1'}
  {attribute 'TcHmiSymbol.Show'}
  avgPower : LREAL;
  {attribute 'OPC.UA.DA' := '1'}
  {attribute 'OPC.UA.DA.Access' := '1'}
  {attribute 'TcHmiSymbol.Show'}
  totalPower : LREAL;
  {attribute 'OPC.UA.DA' := '1'}
  {attribute 'OPC.UA.DA.Access' := '1'}
  {attribute 'TcHmiSymbol.Show'}
  ptpAvgTemp : ARRAY[1..5] OF LREAL;
  {attribute 'OPC.UA.DA' := '1'}
  {attribute 'OPC.UA.DA.Access' := '1'}
  {attribute 'TcHmiSymbol.Show'}
  ptpAllTemp : ARRAY[1..5] OF LREAL;
  {attribute 'OPC.UA.DA' := '1'}
  {attribute 'TcHmiSymbol.Show'}
  stat : ShieldStatuses;
  {attribute 'OPC.UA.DA' := '1'}
  {attribute 'TcHmiSymbol.Show'}
  parts : M_SM_ShieldParts;
  {attribute 'OPC.UA.DA' := '1'}
  {attribute 'TcHmiSymbol.Show'}
  proc : M_SM_ShieldProcesses;
END_STRUCT;
END_TYPE

TYPE M_SM_Bench : STRUCT
  {attribute 'OPC.UA.DA' := '1'}
  {attribute 'OPC.UA.DA.Access' := '1'}
  {attribute 'TcHmiSymbol.Show'}
  actualStatus : STRING;
  {attribute 'OPC.UA.DA' := '1'}
  {attribute 'TcHmiSymbol.Show'}
  stat : BenchStatuses;
  {attribute 'OPC.UA.DA' := '1'}
  {attribute 'TcHmiSymbol.Show'}
  parts : M_SM_BenchParts;
  {attribute 'OPC.UA.DA' := '1'}
  {attribute 'TcHmiSymbol.Show'}
  proc : M_SM_BenchProcesses;
END_STRUCT;
END_TYPE

TYPE M_SM_Cryo : STRUCT
  {attribute 'OPC.UA.DA' := '1'}
  {attribute 'OPC.UA.DA.Access' := '1'}
  {attribute 'TcHmiSymbol.Show'}
  tStatCryoRearOk : BOOL;
  {attribute 'OPC.UA.DA' := '1'}
  {attribute 'OPC.UA.DA.Access' := '1'}
  {attribute 'TcHmiSymbol.Show'}
  actualStatus : STRING;
  {attribute 'OPC.UA.DA' := '1'}
  {attribute 'OPC.UA.DA.Access' := '1'}
  {attribute 'TcHmiSymbol.Show'}
  tStatCryoRearPwr : BOOL;
  {attribute 'OPC.UA.DA' := '1'}
  {attribute 'TcHmiSymbol.Show'}
  stat : CryoStatuses;
  {attribute 'OPC.UA.DA' := '1'}
  {attribute 'TcHmiSymbol.Show'}
  parts : M_SM_CryoParts;
  {attribute 'OPC.UA.DA' := '1'}
  {attribute 'TcHmiSymbol.Show'}
  proc : M_SM_CryoProcesses;
END_STRUCT;
END_TYPE

TYPE M_SM_Thermo : STRUCT
  {attribute 'OPC.UA.DA' := '1'}
  {attribute 'OPC.UA.DA.Access' := '1'}
  {attribute 'TcHmiSymbol.Show'}
  actualStatus : STRING;
  {attribute 'OPC.UA.DA' := '1'}
  {attribute 'TcHmiSymbol.Show'}
  stat : ThermoStatuses;
  {attribute 'OPC.UA.DA' := '1'}
  {attribute 'TcHmiSymbol.Show'}
  parts : M_SM_ThermoParts;
  {attribute 'OPC.UA.DA' := '1'}
  {attribute 'TcHmiSymbol.Show'}
  proc : M_SM_ThermoProcesses;
END_STRUCT;
END_TYPE

TYPE M_SM_Vac : STRUCT
  {attribute 'OPC.UA.DA' := '1'}
  {attribute 'OPC.UA.DA.Access' := '1'}
  {attribute 'TcHmiSymbol.Show'}
  actualStatus : STRING;
  {attribute 'OPC.UA.DA' := '1'}
  {attribute 'TcHmiSymbol.Show'}
  stat : VacStatuses;
  {attribute 'OPC.UA.DA' := '1'}
  {attribute 'TcHmiSymbol.Show'}
  proc : M_SM_VacProcesses;
END_STRUCT;
END_TYPE

TYPE M_SM_ThermoVac : STRUCT
  {attribute 'OPC.UA.DA' := '1'}
  {attribute 'OPC.UA.DA.Access' := '3'}
  {attribute 'TcHmiSymbol.Show'}
  editableConfig : ThermoVacConfig;
  {attribute 'OPC.UA.DA' := '1'}
  {attribute 'OPC.UA.DA.Access' := '1'}
  {attribute 'TcHmiSymbol.Show'}
  actualStatus : STRING;
  {attribute 'OPC.UA.DA' := '1'}
  {attribute 'OPC.UA.DA.Access' := '1'}
  {attribute 'TcHmiSymbol.Show'}
  config : ThermoVacConfig;
  {attribute 'OPC.UA.DA' := '1'}
  {attribute 'TcHmiSymbol.Show'}
  stat : ThermoVacStatuses;
  {attribute 'OPC.UA.DA' := '1'}
  {attribute 'TcHmiSymbol.Show'}
  parts : M_SM_ThermoVacParts;
  {attribute 'OPC.UA.DA' := '1'}
  {attribute 'TcHmiSymbol.Show'}
  proc : M_SM_ThermoVacProcesses;
END_STRUCT;
END_TYPE

TYPE M_ForceHeater : STRUCT
  {attribute 'OPC.UA.DA' := '1'}
  {attribute 'OPC.UA.DA.Access' := '3'}
  {attribute 'TcHmiSymbol.Show'}
  set : ForceHeaterArgs;
END_STRUCT;
END_TYPE

TYPE M_SM_TempMeasurementProcesses : STRUCT
  {attribute 'TcHmiSymbol.Show'}
  initialize : M_Process;
  {attribute 'TcHmiSymbol.Show'}
  clearPtp : M_Process;
END_STRUCT;
END_TYPE

TYPE M_SM_HeaterProcesses : STRUCT
  {attribute 'TcHmiSymbol.Show'}
  initialize : M_Process;
  {attribute 'TcHmiSymbol.Show'}
  reset : M_Process;
  {attribute 'TcHmiSymbol.Show'}
  force : M_ForceHeater;
END_STRUCT;
END_TYPE

TYPE M_SM_OuterRoomParts : STRUCT
  {attribute 'TcHmiSymbol.Show'}
  tFloorE : M_TempMeasurement;
  {attribute 'TcHmiSymbol.Show'}
  tFloorW : M_TempMeasurement;
  {attribute 'TcHmiSymbol.Show'}
  tTopN : M_TempMeasurement;
  {attribute 'TcHmiSymbol.Show'}
  tTopS : M_TempMeasurement;
  {attribute 'TcHmiSymbol.Show'}
  ref : M_RefSensor;
END_STRUCT;
END_TYPE

TYPE M_SM_OuterRoomProcesses : STRUCT
  {attribute 'TcHmiSymbol.Show'}
  initialize : M_Process;
  {attribute 'TcHmiSymbol.Show'}
  start : M_Process;
  {attribute 'TcHmiSymbol.Show'}
  stop : M_Process;
  {attribute 'TcHmiSymbol.Show'}
  reset : M_Process;
  {attribute 'TcHmiSymbol.Show'}
  clearPtp : M_Process;
  {attribute 'TcHmiSymbol.Show'}
  lock : M_Process;
  {attribute 'TcHmiSymbol.Show'}
  unlock : M_Process;
END_STRUCT;
END_TYPE

TYPE M_SM_InnerRoomParts : STRUCT
  {attribute 'TcHmiSymbol.Show'}
  tAbove : M_TempMeasurement;
  {attribute 'TcHmiSymbol.Show'}
  tBelow : M_TempMeasurement;
  {attribute 'TcHmiSymbol.Show'}
  tEast : M_TempMeasurement;
  {attribute 'TcHmiSymbol.Show'}
  tWest : M_TempMeasurement;
  {attribute 'TcHmiSymbol.Show'}
  htDucts : M_Heater;
  {attribute 'TcHmiSymbol.Show'}
  ref : M_RefSensor;
END_STRUCT;
END_TYPE

TYPE M_SM_InnerRoomProcesses : STRUCT
  {attribute 'TcHmiSymbol.Show'}
  initialize : M_Process;
  {attribute 'TcHmiSymbol.Show'}
  start : M_Process;
  {attribute 'TcHmiSymbol.Show'}
  stop : M_Process;
  {attribute 'TcHmiSymbol.Show'}
  reset : M_Process;
  {attribute 'TcHmiSymbol.Show'}
  clearPtp : M_Process;
  {attribute 'TcHmiSymbol.Show'}
  lock : M_Process;
  {attribute 'TcHmiSymbol.Show'}
  unlock : M_Process;
END_STRUCT;
END_TYPE

TYPE M_SM_VesselParts : STRUCT
  {attribute 'TcHmiSymbol.Show'}
  tLegNE : M_TempMeasurement;
  {attribute 'TcHmiSymbol.Show'}
  tLegNW : M_TempMeasurement;
  {attribute 'TcHmiSymbol.Show'}
  tLegSE : M_TempMeasurement;
  {attribute 'TcHmiSymbol.Show'}
  tLegSW : M_TempMeasurement;
  {attribute 'TcHmiSymbol.Show'}
  tLegTopNE : M_TempMeasurement;
  {attribute 'TcHmiSymbol.Show'}
  tLegTopNW : M_TempMeasurement;
  {attribute 'TcHmiSymbol.Show'}
  tLegTopSE : M_TempMeasurement;
  {attribute 'TcHmiSymbol.Show'}
  tLegTopSW : M_TempMeasurement;
  {attribute 'TcHmiSymbol.Show'}
  tBotNE : M_TempMeasurement;
  {attribute 'TcHmiSymbol.Show'}
  tBotNW : M_TempMeasurement;
  {attribute 'TcHmiSymbol.Show'}
  tBotSE : M_TempMeasurement;
  {attribute 'TcHmiSymbol.Show'}
  tBotSW : M_TempMeasurement;
  {attribute 'TcHmiSymbol.Show'}
  tCenter : M_TempMeasurement;
  {attribute 'TcHmiSymbol.Show'}
  tCenterTH10K : M_TempMeasurement;
  {attribute 'TcHmiSymbol.Show'}
  tSideN : M_TempMeasurement;
  {attribute 'TcHmiSymbol.Show'}
  tSideS : M_TempMeasurement;
  {attribute 'TcHmiSymbol.Show'}
  tSideE : M_TempMeasurement;
  {attribute 'TcHmiSymbol.Show'}
  tSideW : M_TempMeasurement;
  {attribute 'TcHmiSymbol.Show'}
  tLidN : M_TempMeasurement;
  {attribute 'TcHmiSymbol.Show'}
  tLidS : M_TempMeasurement;
  {attribute 'TcHmiSymbol.Show'}
  htLegNE : M_Heater;
  {attribute 'TcHmiSymbol.Show'}
  htLegNW : M_Heater;
  {attribute 'TcHmiSymbol.Show'}
  htLegSE : M_Heater;
  {attribute 'TcHmiSymbol.Show'}
  htLegSW : M_Heater;
  {attribute 'TcHmiSymbol.Show'}
  htLegTopNE : M_Heater;
  {attribute 'TcHmiSymbol.Show'}
  htLegTopNW : M_Heater;
  {attribute 'TcHmiSymbol.Show'}
  htLegTopSE : M_Heater;
  {attribute 'TcHmiSymbol.Show'}
  htLegTopSW : M_Heater;
  {attribute 'TcHmiSymbol.Show'}
  htBotNE : M_Heater;
  {attribute 'TcHmiSymbol.Show'}
  htBotNW : M_Heater;
  {attribute 'TcHmiSymbol.Show'}
  htBotSE : M_Heater;
  {attribute 'TcHmiSymbol.Show'}
  htBotSW : M_Heater;
  {attribute 'TcHmiSymbol.Show'}
  htSideN : M_Heater;
  {attribute 'TcHmiSymbol.Show'}
  htSideS : M_Heater;
  {attribute 'TcHmiSymbol.Show'}
  htSideE : M_Heater;
  {attribute 'TcHmiSymbol.Show'}
  htSideW : M_Heater;
  {attribute 'TcHmiSymbol.Show'}
  htLidN : M_Heater;
  {attribute 'TcHmiSymbol.Show'}
  htLidS : M_Heater;
  {attribute 'TcHmiSymbol.Show'}
  ref : M_RefSensor;
END_STRUCT;
END_TYPE

TYPE M_SM_VesselProcesses : STRUCT
  {attribute 'TcHmiSymbol.Show'}
  initialize : M_Process;
  {attribute 'TcHmiSymbol.Show'}
  start : M_Process;
  {attribute 'TcHmiSymbol.Show'}
  stop : M_Process;
  {attribute 'TcHmiSymbol.Show'}
  reset : M_Process;
  {attribute 'TcHmiSymbol.Show'}
  clearPtp : M_Process;
  {attribute 'TcHmiSymbol.Show'}
  lock : M_Process;
  {attribute 'TcHmiSymbol.Show'}
  unlock : M_Process;
END_STRUCT;
END_TYPE

TYPE M_SM_ShieldParts : STRUCT
  {attribute 'TcHmiSymbol.Show'}
  tTopNE : M_TempMeasurement;
  {attribute 'TcHmiSymbol.Show'}
  tTopNW : M_TempMeasurement;
  {attribute 'TcHmiSymbol.Show'}
  tTopSE : M_TempMeasurement;
  {attribute 'TcHmiSymbol.Show'}
  tTopSW : M_TempMeasurement;
  {attribute 'TcHmiSymbol.Show'}
  tSideN : M_TempMeasurement;
  {attribute 'TcHmiSymbol.Show'}
  tSideS : M_TempMeasurement;
  {attribute 'TcHmiSymbol.Show'}
  tSideNE : M_TempMeasurement;
  {attribute 'TcHmiSymbol.Show'}
  tSideSE : M_TempMeasurement;
  {attribute 'TcHmiSymbol.Show'}
  tSideNW : M_TempMeasurement;
  {attribute 'TcHmiSymbol.Show'}
  tSideSW : M_TempMeasurement;
  {attribute 'TcHmiSymbol.Show'}
  tBotNE : M_TempMeasurement;
  {attribute 'TcHmiSymbol.Show'}
  tBotNW : M_TempMeasurement;
  {attribute 'TcHmiSymbol.Show'}
  tBotS : M_TempMeasurement;
  {attribute 'TcHmiSymbol.Show'}
  tCentre : M_TempMeasurement;
  {attribute 'TcHmiSymbol.Show'}
  tCentreTh10k : M_TempMeasurement;
  {attribute 'TcHmiSymbol.Show'}
  htTopNE : M_Heater;
  {attribute 'TcHmiSymbol.Show'}
  htTopNW : M_Heater;
  {attribute 'TcHmiSymbol.Show'}
  htTopSE : M_Heater;
  {attribute 'TcHmiSymbol.Show'}
  htTopSW : M_Heater;
  {attribute 'TcHmiSymbol.Show'}
  htSideN : M_Heater;
  {attribute 'TcHmiSymbol.Show'}
  htSideS : M_Heater;
  {attribute 'TcHmiSymbol.Show'}
  htSideNE : M_Heater;
  {attribute 'TcHmiSymbol.Show'}
  htSideSE : M_Heater;
  {attribute 'TcHmiSymbol.Show'}
  htSideNW : M_Heater;
  {attribute 'TcHmiSymbol.Show'}
  htSideSW : M_Heater;
  {attribute 'TcHmiSymbol.Show'}
  htBotNE : M_Heater;
  {attribute 'TcHmiSymbol.Show'}
  htBotNW : M_Heater;
  {attribute 'TcHmiSymbol.Show'}
  htBotS : M_Heater;
  {attribute 'TcHmiSymbol.Show'}
  htCentre : M_Heater;
  {attribute 'TcHmiSymbol.Show'}
  ref : M_RefSensor;
END_STRUCT;
END_TYPE

TYPE M_SM_ShieldProcesses : STRUCT
  {attribute 'TcHmiSymbol.Show'}
  initialize : M_Process;
  {attribute 'TcHmiSymbol.Show'}
  start : M_Process;
  {attribute 'TcHmiSymbol.Show'}
  stop : M_Process;
  {attribute 'TcHmiSymbol.Show'}
  reset : M_Process;
  {attribute 'TcHmiSymbol.Show'}
  clearPtp : M_Process;
  {attribute 'TcHmiSymbol.Show'}
  lock : M_Process;
  {attribute 'TcHmiSymbol.Show'}
  unlock : M_Process;
END_STRUCT;
END_TYPE

TYPE M_SM_BenchParts : STRUCT
  {attribute 'TcHmiSymbol.Show'}
  tCentre : M_TempMeasurement;
  {attribute 'TcHmiSymbol.Show'}
  tCentreTH10k : M_TempMeasurement;
  {attribute 'TcHmiSymbol.Show'}
  tCollBench : M_TempMeasurement;
  {attribute 'TcHmiSymbol.Show'}
  tEchelleCryo : M_TempMeasurement;
  {attribute 'TcHmiSymbol.Show'}
  tCamCryo : M_TempMeasurement;
  {attribute 'TcHmiSymbol.Show'}
  tColl : M_TempMeasurement;
  {attribute 'TcHmiSymbol.Show'}
  tPrism : M_TempMeasurement;
  {attribute 'TcHmiSymbol.Show'}
  tEchelle : M_TempMeasurement;
  {attribute 'TcHmiSymbol.Show'}
  tCam : M_TempMeasurement;
  {attribute 'TcHmiSymbol.Show'}
  tInOptics : M_TempMeasurement;
  {attribute 'TcHmiSymbol.Show'}
  htCollBench : M_Heater;
  {attribute 'TcHmiSymbol.Show'}
  htEchelleCryo : M_Heater;
  {attribute 'TcHmiSymbol.Show'}
  htCamCryo : M_Heater;
  {attribute 'TcHmiSymbol.Show'}
  htEchellePrism : M_Heater;
  {attribute 'TcHmiSymbol.Show'}
  ref : M_RefSensor;
END_STRUCT;
END_TYPE

TYPE M_SM_BenchProcesses : STRUCT
  {attribute 'TcHmiSymbol.Show'}
  initialize : M_Process;
  {attribute 'TcHmiSymbol.Show'}
  start : M_Process;
  {attribute 'TcHmiSymbol.Show'}
  stop : M_Process;
  {attribute 'TcHmiSymbol.Show'}
  reset : M_Process;
  {attribute 'TcHmiSymbol.Show'}
  clearPtp : M_Process;
  {attribute 'TcHmiSymbol.Show'}
  lock : M_Process;
  {attribute 'TcHmiSymbol.Show'}
  unlock : M_Process;
END_STRUCT;
END_TYPE

TYPE M_SM_CryoParts : STRUCT
  {attribute 'TcHmiSymbol.Show'}
  tRearOut : M_TempMeasurement;
  {attribute 'TcHmiSymbol.Show'}
  tRearIn : M_TempMeasurement;
  {attribute 'TcHmiSymbol.Show'}
  tFront : M_TempMeasurement;
  {attribute 'TcHmiSymbol.Show'}
  htRearOut : M_Heater;
  {attribute 'TcHmiSymbol.Show'}
  htRearIn : M_Heater;
  {attribute 'TcHmiSymbol.Show'}
  htRearFront : M_Heater;
  {attribute 'TcHmiSymbol.Show'}
  ref : M_RefSensor;
END_STRUCT;
END_TYPE

TYPE M_SM_CryoProcesses : STRUCT
  {attribute 'TcHmiSymbol.Show'}
  initialize : M_Process;
  {attribute 'TcHmiSymbol.Show'}
  start : M_Process;
  {attribute 'TcHmiSymbol.Show'}
  stop : M_Process;
  {attribute 'TcHmiSymbol.Show'}
  reset : M_Process;
  {attribute 'TcHmiSymbol.Show'}
  clearPtp : M_Process;
  {attribute 'TcHmiSymbol.Show'}
  lock : M_Process;
  {attribute 'TcHmiSymbol.Show'}
  unlock : M_Process;
END_STRUCT;
END_TYPE

TYPE M_SM_ThermoParts : STRUCT
  {attribute 'TcHmiSymbol.Show'}
  outerRoom : M_OuterRoom;
  {attribute 'TcHmiSymbol.Show'}
  innerRoom : M_InnerRoom;
  {attribute 'TcHmiSymbol.Show'}
  vessel : M_Vessel;
  {attribute 'TcHmiSymbol.Show'}
  shield : M_Shield;
  {attribute 'TcHmiSymbol.Show'}
  bench : M_Bench;
  {attribute 'TcHmiSymbol.Show'}
  cryo : M_Cryo;
END_STRUCT;
END_TYPE

TYPE M_SM_ThermoProcesses : STRUCT
  {attribute 'TcHmiSymbol.Show'}
  initialize : M_Process;
  {attribute 'TcHmiSymbol.Show'}
  start : M_Process;
  {attribute 'TcHmiSymbol.Show'}
  stop : M_Process;
  {attribute 'TcHmiSymbol.Show'}
  clearPtp : M_Process;
  {attribute 'TcHmiSymbol.Show'}
  reset : M_Process;
  {attribute 'TcHmiSymbol.Show'}
  lock : M_Process;
  {attribute 'TcHmiSymbol.Show'}
  unlock : M_Process;
END_STRUCT;
END_TYPE

TYPE M_SM_VacProcesses : STRUCT
  {attribute 'TcHmiSymbol.Show'}
  initialize : M_Process;
  {attribute 'TcHmiSymbol.Show'}
  reset : M_Process;
  {attribute 'TcHmiSymbol.Show'}
  lock : M_Process;
  {attribute 'TcHmiSymbol.Show'}
  unlock : M_Process;
END_STRUCT;
END_TYPE

TYPE M_SM_ThermoVacParts : STRUCT
  {attribute 'TcHmiSymbol.Show'}
  thermo : M_Thermo;
  {attribute 'TcHmiSymbol.Show'}
  vac : M_Vac;
  {attribute 'TcHmiSymbol.Show'}
  configManager : M_ConfigManager;
END_STRUCT;
END_TYPE

TYPE M_SM_ThermoVacProcesses : STRUCT
  {attribute 'TcHmiSymbol.Show'}
  initialize : M_Process;
  {attribute 'TcHmiSymbol.Show'}
  reset : M_Process;
  {attribute 'TcHmiSymbol.Show'}
  lock : M_Process;
  {attribute 'TcHmiSymbol.Show'}
  unlock : M_Process;
END_STRUCT;
END_TYPE

{attribute 'TcRpcEnable' := '1'}
FUNCTION F_TempControlStatus : TempControlStatus
  VAR_INPUT
    superState : BOOL := TRUE;  (* Super state (TRUE if the super state is active, or if there is no super state) *)
    isActive : BOOL;  (* True if the temp control is active (not idle) *)
    isWarmingUp : BOOL;  (* True if the system warming up *)
  END_VAR

              IF NOT(superState) THEN
    F_TempControlStatus := TempControlStatus.unknown;
ELSIF (NOT(isActive)) AND (NOT(isWarmingUp)) THEN
    F_TempControlStatus := TempControlStatus.idle;
ELSIF isWarmingUp THEN
    F_TempControlStatus := TempControlStatus.warming_up;
ELSIF isActive AND (NOT(isWarmingUp)) THEN
    F_TempControlStatus := TempControlStatus.active;
ELSE
    F_TempControlStatus := TempControlStatus.invalid_model;
END_IF;

            
END_FUNCTION

FUNCTION_BLOCK SM_RefSensor
  VAR_OUTPUT
    {attribute 'OPC.UA.DA' := '1'}
    {attribute 'OPC.UA.DA.Access' := '1'}
    actualStatus : STRING(50);  (* Current status description *)
    {attribute 'OPC.UA.DA' := '1'}
    {attribute 'OPC.UA.DA.Access' := '1'}
    value : LREAL;  (* Measured value *)
  END_VAR

            
          

METHOD _copyFromModel_SM_RefSensor
  VAR_IN_OUT
    {attribute 'OPC.UA.DA' := '0'}
    model : M_SM_RefSensor;
  END_VAR
                  
                
END_METHOD

METHOD _copyToModel_SM_RefSensor
  VAR_IN_OUT
    {attribute 'OPC.UA.DA' := '0'}
    model : M_SM_RefSensor;
  END_VAR
                  model.actualStatus := THIS^.actualStatus;
model.value := THIS^.value;

                
END_METHOD
END_FUNCTION_BLOCK

FUNCTION_BLOCK SM_TempMeasurement
  VAR_INPUT
    {attribute 'OPC.UA.DA' := '1'}
    {attribute 'OPC.UA.DA.Access' := '1'}
    isSimulated : BOOL;
    {attribute 'OPC.UA.DA' := '0'}
    rawValue AT %I* : REAL;  (* Raw measured value *)
    {attribute 'OPC.UA.DA' := '0'}
    error : BOOL;  (* True if sensor error *)
  END_VAR
  VAR_OUTPUT
    {attribute 'OPC.UA.DA' := '1'}
    {attribute 'OPC.UA.DA.Access' := '1'}
    actualStatus : STRING(50);  (* Current status description *)
    {attribute 'OPC.UA.DA' := '1'}
    {attribute 'OPC.UA.DA.Access' := '1'}
    value : LREAL;  (* Measured value *)
    {attribute 'OPC.UA.DA' := '1'}
    {attribute 'OPC.UA.DA.Access' := '1'}
    ptp1 : LREAL;
    {attribute 'OPC.UA.DA' := '1'}
    {attribute 'OPC.UA.DA.Access' := '1'}
    ptp2 : LREAL;
    {attribute 'OPC.UA.DA' := '1'}
    stat : TempMeasurementStatuses;  (* Statuses of the state machine *)
    {attribute 'OPC.UA.DA' := '1'}
    proc : TempMeasurementProcesses;  (* Processes of the state machine *)
  END_VAR
  VAR_IN_OUT
    {attribute 'OPC.UA.DA' := '0'}
    config_ref : MeasurementConfig2;  (* Reference to the config *)
    {attribute 'OPC.UA.DA' := '0'}
    sharedConfig_ref : SharedMeasurementConfig;  (* Reference to sensor alarm config *)
  END_VAR

            stat.enabled := F_EnabledStatus(
    superState := TRUE,
    isEnabled := config_ref.enabled);
stat.health := F_HealthStatus(
    superState := stat.enabled = EnabledStatus.enabled,
    isGood := NOT((stat.alarm = HiHiLoLoAlarmStatus.hiHi) OR ((stat.alarm = HiHiLoLoAlarmStatus.loLo) OR error)),
    hasWarning := (stat.alarm = HiHiLoLoAlarmStatus.hi) OR ((stat.alarm = HiHiLoLoAlarmStatus.lo) OR (NOT(sharedConfig_ref.alarms.enabled))));
proc.initialize( isEnabled := NOT((stat.init = InitializationStatus.locked) OR (stat.enabled = EnabledStatus.disabled)) );
proc.clearPtp( isEnabled := stat.init = InitializationStatus.initialized );

          

METHOD _copyFromModel_SM_TempMeasurement
  VAR_IN_OUT
    {attribute 'OPC.UA.DA' := '0'}
    model : M_SM_TempMeasurement;
  END_VAR
                  THIS^.proc.initialize._copyFromModel_Process( model := model.proc.initialize );
THIS^.proc.clearPtp._copyFromModel_Process( model := model.proc.clearPtp );

                
END_METHOD

METHOD _copyToModel_SM_TempMeasurement
  VAR_IN_OUT
    {attribute 'OPC.UA.DA' := '0'}
    model : M_SM_TempMeasurement;
  END_VAR
                  model.isSimulated := THIS^.isSimulated;
model.actualStatus := THIS^.actualStatus;
model.value := THIS^.value;
model.ptp1 := THIS^.ptp1;
model.ptp2 := THIS^.ptp2;
model.stat := THIS^.stat;
THIS^.proc.initialize._copyToModel_Process( model := model.proc.initialize );
THIS^.proc.clearPtp._copyToModel_Process( model := model.proc.clearPtp );

                
END_METHOD
END_FUNCTION_BLOCK

FUNCTION_BLOCK SM_Heater
  VAR_INPUT
    {attribute 'OPC.UA.DA' := '1'}
    {attribute 'OPC.UA.DA.Access' := '1'}
    setPoint : LREAL;  (* Current set point of the heater in kelvin *)
    {attribute 'OPC.UA.DA' := '1'}
    {attribute 'OPC.UA.DA.Access' := '1'}
    temp : LREAL;  (* Associated temperature of the heater in kelvin *)
    {attribute 'OPC.UA.DA' := '1'}
    {attribute 'OPC.UA.DA.Access' := '1'}
    isSimulated : BOOL;
  END_VAR
  VAR_OUTPUT
    {attribute 'OPC.UA.DA' := '1'}
    {attribute 'OPC.UA.DA.Access' := '1'}
    actualStatus : STRING(50);  (* Current status description *)
    {attribute 'OPC.UA.DA' := '1'}
    {attribute 'OPC.UA.DA.Access' := '1'}
    power : LREAL;  (* Current power of the heater in percentage *)
    {attribute 'OPC.UA.DA' := '1'}
    {attribute 'OPC.UA.DA.Access' := '1'}
    deviation : LREAL;  (* Current error between set point and associated temperature *)
    {attribute 'OPC.UA.DA' := '1'}
    {attribute 'OPC.UA.DA.Access' := '1'}
    isForced : BOOL;  (* True if the heater power is forced (overwriting the normal control) *)
    {attribute 'OPC.UA.DA' := '1'}
    {attribute 'OPC.UA.DA.Access' := '1'}
    simTemp : LREAL;  (* Simulated temperature for testing the heater control *)
    {attribute 'OPC.UA.DA' := '1'}
    stat : HeaterStatuses;  (* Statuses of the state machine *)
    {attribute 'OPC.UA.DA' := '1'}
    proc : HeaterProcesses;  (* Processes of the state machine *)
  END_VAR
  VAR_IN_OUT
    {attribute 'OPC.UA.DA' := '0'}
    config_ref : HeaterConfig;  (* Reference to the heater config *)
    {attribute 'OPC.UA.DA' := '0'}
    sharedConfig_ref : SharedHeaterConfig;  (* Reference to the shared heater config *)
    {attribute 'OPC.UA.DA' := '0'}
    operator_ref : OperatorStatus;  (* Shared operator status *)
  END_VAR

            stat.enabled := F_EnabledStatus(
    superState := TRUE,
    isEnabled := config_ref.enabled);
proc.initialize( isEnabled := NOT((stat.init = InitializationStatus.locked) OR (stat.init = InitializationStatus.initializing)) );
proc.reset( isEnabled := TRUE );
proc.force( isEnabled := (operator_ref = OperatorStatus.tech) AND ((NOT(isForced)) AND ((stat.enabled = EnabledStatus.enabled) AND (stat.init = InitializationStatus.initialized))) );

          

METHOD _copyFromModel_SM_Heater
  VAR_IN_OUT
    {attribute 'OPC.UA.DA' := '0'}
    model : M_SM_Heater;
  END_VAR
                  THIS^.proc.initialize._copyFromModel_Process( model := model.proc.initialize );
THIS^.proc.reset._copyFromModel_Process( model := model.proc.reset );
THIS^.proc.force._copyFromModel_ForceHeater( model := model.proc.force );

                
END_METHOD

METHOD _copyToModel_SM_Heater
  VAR_IN_OUT
    {attribute 'OPC.UA.DA' := '0'}
    model : M_SM_Heater;
  END_VAR
                  model.setPoint := THIS^.setPoint;
model.temp := THIS^.temp;
model.isSimulated := THIS^.isSimulated;
model.actualStatus := THIS^.actualStatus;
model.power := THIS^.power;
model.deviation := THIS^.deviation;
model.isForced := THIS^.isForced;
model.simTemp := THIS^.simTemp;
model.stat := THIS^.stat;
THIS^.proc.initialize._copyToModel_Process( model := model.proc.initialize );
THIS^.proc.reset._copyToModel_Process( model := model.proc.reset );
THIS^.proc.force._copyToModel_ForceHeater( model := model.proc.force );

                
END_METHOD
END_FUNCTION_BLOCK

FUNCTION_BLOCK SM_OuterRoom
  VAR_OUTPUT
    {attribute 'OPC.UA.DA' := '1'}
    {attribute 'OPC.UA.DA.Access' := '1'}
    actualStatus : STRING(50);  (* Current status description *)
    {attribute 'OPC.UA.DA' := '1'}
    stat : OuterRoomStatuses;  (* Statuses of the state machine *)
    {attribute 'OPC.UA.DA' := '1'}
    parts : OuterRoomParts;  (* Parts of the state machine *)
    {attribute 'OPC.UA.DA' := '1'}
    proc : OuterRoomProcesses;  (* Processes of the state machine *)
  END_VAR
  VAR_IN_OUT
    {attribute 'OPC.UA.DA' := '0'}
    config_ref : OuterRoomConfig;  (* Active configuration of the outer room *)
    {attribute 'OPC.UA.DA' := '0'}
    sharedConfig_ref : ThermoSharedConfig;  (* Shared config for the thermo system *)
    {attribute 'OPC.UA.DA' := '0'}
    activity_ref : ActivityStatus;  (* Shared activity status *)
    {attribute 'OPC.UA.DA' := '0'}
    services_ref : Services;  (* Shared services *)
    {attribute 'OPC.UA.DA' := '0'}
    operator_ref : OperatorStatus;  (* Shared operator status *)
  END_VAR

            parts.tFloorE(
    config_ref := config_ref.tFloorE,
    sharedConfig_ref := config_ref.shared.sensors);
parts.tFloorW(
    config_ref := config_ref.tFloorW,
    sharedConfig_ref := config_ref.shared.sensors);
parts.tTopN(
    config_ref := config_ref.tTopN,
    sharedConfig_ref := config_ref.shared.sensors);
parts.tTopS(
    config_ref := config_ref.tTopS,
    sharedConfig_ref := config_ref.shared.sensors);
parts.ref();
stat.enabled := F_EnabledStatus(
    superState := TRUE,
    isEnabled := config_ref.enabled);
stat.busy := F_BusyStatus(
    superState := TRUE,
    isBusy := (stat.control = TempControlStatus.warming_up) OR (stat.init = InitializationStatus.initializing));
proc.initialize();
proc.start();
proc.stop();
proc.reset();
proc.clearPtp();
proc.lock();
proc.unlock();

          

METHOD _copyFromModel_SM_OuterRoom
  VAR_IN_OUT
    {attribute 'OPC.UA.DA' := '0'}
    model : M_SM_OuterRoom;
  END_VAR
                  THIS^.parts.tFloorE._copyFromModel_TempMeasurement( model := model.parts.tFloorE );
THIS^.parts.tFloorW._copyFromModel_TempMeasurement( model := model.parts.tFloorW );
THIS^.parts.tTopN._copyFromModel_TempMeasurement( model := model.parts.tTopN );
THIS^.parts.tTopS._copyFromModel_TempMeasurement( model := model.parts.tTopS );
THIS^.parts.ref._copyFromModel_RefSensor( model := model.parts.ref );
THIS^.proc.initialize._copyFromModel_Process( model := model.proc.initialize );
THIS^.proc.start._copyFromModel_Process( model := model.proc.start );
THIS^.proc.stop._copyFromModel_Process( model := model.proc.stop );
THIS^.proc.reset._copyFromModel_Process( model := model.proc.reset );
THIS^.proc.clearPtp._copyFromModel_Process( model := model.proc.clearPtp );
THIS^.proc.lock._copyFromModel_Process( model := model.proc.lock );
THIS^.proc.unlock._copyFromModel_Process( model := model.proc.unlock );

                
END_METHOD

METHOD _copyToModel_SM_OuterRoom
  VAR_IN_OUT
    {attribute 'OPC.UA.DA' := '0'}
    model : M_SM_OuterRoom;
  END_VAR
                  model.actualStatus := THIS^.actualStatus;
model.stat := THIS^.stat;
THIS^.parts.tFloorE._copyToModel_TempMeasurement( model := model.parts.tFloorE );
THIS^.parts.tFloorW._copyToModel_TempMeasurement( model := model.parts.tFloorW );
THIS^.parts.tTopN._copyToModel_TempMeasurement( model := model.parts.tTopN );
THIS^.parts.tTopS._copyToModel_TempMeasurement( model := model.parts.tTopS );
THIS^.parts.ref._copyToModel_RefSensor( model := model.parts.ref );
THIS^.proc.initialize._copyToModel_Process( model := model.proc.initialize );
THIS^.proc.start._copyToModel_Process( model := model.proc.start );
THIS^.proc.stop._copyToModel_Process( model := model.proc.stop );
THIS^.proc.reset._copyToModel_Process( model := model.proc.reset );
THIS^.proc.clearPtp._copyToModel_Process( model := model.proc.clearPtp );
THIS^.proc.lock._copyToModel_Process( model := model.proc.lock );
THIS^.proc.unlock._copyToModel_Process( model := model.proc.unlock );

                
END_METHOD
END_FUNCTION_BLOCK

FUNCTION_BLOCK SM_InnerRoom
  VAR_OUTPUT
    {attribute 'OPC.UA.DA' := '1'}
    {attribute 'OPC.UA.DA.Access' := '1'}
    actualStatus : STRING(50);  (* Current status description *)
    {attribute 'OPC.UA.DA' := '1'}
    {attribute 'OPC.UA.DA.Access' := '1'}
    setPoint : LREAL;  (* The ramped setpoint used by the pid *)
    {attribute 'OPC.UA.DA' := '1'}
    {attribute 'OPC.UA.DA.Access' := '1'}
    avgTemp : LREAL;  (* Average temperature of the vessel in kelvin *)
    {attribute 'OPC.UA.DA' := '1'}
    {attribute 'OPC.UA.DA.Access' := '1'}
    avgPower : LREAL;  (* Average power of the heaters in percentage *)
    {attribute 'OPC.UA.DA' := '1'}
    {attribute 'OPC.UA.DA.Access' := '1'}
    totalPower : LREAL;  (* Total power of all heaters in watt *)
    {attribute 'OPC.UA.DA' := '1'}
    {attribute 'OPC.UA.DA.Access' := '1'}
    ptpAvgTemp : ARRAY[1..5] OF LREAL;  (* ptp values of the average temperature of the vessel" *)
    {attribute 'OPC.UA.DA' := '1'}
    {attribute 'OPC.UA.DA.Access' := '1'}
    ptpAllTemp : ARRAY[1..5] OF LREAL;  (* ptp values of all temp measurements in the vessel" *)
    {attribute 'OPC.UA.DA' := '1'}
    stat : InnerRoomStatuses;  (* Statuses of the state machine *)
    {attribute 'OPC.UA.DA' := '1'}
    parts : InnerRoomParts;  (* Parts of the state machine *)
    {attribute 'OPC.UA.DA' := '1'}
    proc : InnerRoomProcesses;  (* Processes of the state machine *)
  END_VAR
  VAR_IN_OUT
    {attribute 'OPC.UA.DA' := '0'}
    config_ref : InnerRoomConfig;  (* Active configuration of the inner room *)
    {attribute 'OPC.UA.DA' := '0'}
    sharedConfig_ref : ThermoSharedConfig;  (* Shared config for the thermo system *)
    {attribute 'OPC.UA.DA' := '0'}
    activity_ref : ActivityStatus;  (* Shared activity status *)
    {attribute 'OPC.UA.DA' := '0'}
    services_ref : Services;  (* Shared services *)
    {attribute 'OPC.UA.DA' := '0'}
    operator_ref : OperatorStatus;  (* Shared operator status *)
  END_VAR

            parts.tAbove(
    config_ref := config_ref.tAbove,
    sharedConfig_ref := config_ref.shared.sensors);
parts.tBelow(
    config_ref := config_ref.tBelow,
    sharedConfig_ref := config_ref.shared.sensors);
parts.tEast(
    config_ref := config_ref.tEast,
    sharedConfig_ref := config_ref.shared.sensors);
parts.tWest(
    config_ref := config_ref.tWest,
    sharedConfig_ref := config_ref.shared.sensors);
parts.htDucts(
    config_ref := config_ref.htDucts,
    sharedConfig_ref := config_ref.shared.heaters,
    operator_ref := operator_ref);
parts.ref();
stat.enabled := F_EnabledStatus(
    superState := TRUE,
    isEnabled := config_ref.enabled);
stat.busy := F_BusyStatus(
    superState := TRUE,
    isBusy := (stat.control = TempControlStatus.warming_up) OR (stat.init = InitializationStatus.initializing));
proc.initialize( isEnabled := NOT((stat.init = InitializationStatus.locked) OR (stat.enabled = EnabledStatus.disabled)) );
proc.start( isEnabled := (stat.control = TempControlStatus.idle) AND ((stat.init = InitializationStatus.initialized) AND (stat.enabled = EnabledStatus.enabled)) );
proc.stop( isEnabled := (NOT(stat.control = TempControlStatus.idle)) AND (stat.init = InitializationStatus.initialized) );
proc.reset( isEnabled := TRUE );
proc.clearPtp( isEnabled := (operator_ref = OperatorStatus.tech) AND (stat.init = InitializationStatus.initialized) );
proc.lock( isEnabled := (operator_ref = OperatorStatus.tech) AND (NOT(stat.init = InitializationStatus.locked)) );
proc.unlock( isEnabled := (operator_ref = OperatorStatus.tech) AND (stat.init = InitializationStatus.locked) );

          

METHOD _copyFromModel_SM_InnerRoom
  VAR_IN_OUT
    {attribute 'OPC.UA.DA' := '0'}
    model : M_SM_InnerRoom;
  END_VAR
                  THIS^.parts.tAbove._copyFromModel_TempMeasurement( model := model.parts.tAbove );
THIS^.parts.tBelow._copyFromModel_TempMeasurement( model := model.parts.tBelow );
THIS^.parts.tEast._copyFromModel_TempMeasurement( model := model.parts.tEast );
THIS^.parts.tWest._copyFromModel_TempMeasurement( model := model.parts.tWest );
THIS^.parts.htDucts._copyFromModel_Heater( model := model.parts.htDucts );
THIS^.parts.ref._copyFromModel_RefSensor( model := model.parts.ref );
THIS^.proc.initialize._copyFromModel_Process( model := model.proc.initialize );
THIS^.proc.start._copyFromModel_Process( model := model.proc.start );
THIS^.proc.stop._copyFromModel_Process( model := model.proc.stop );
THIS^.proc.reset._copyFromModel_Process( model := model.proc.reset );
THIS^.proc.clearPtp._copyFromModel_Process( model := model.proc.clearPtp );
THIS^.proc.lock._copyFromModel_Process( model := model.proc.lock );
THIS^.proc.unlock._copyFromModel_Process( model := model.proc.unlock );

                
END_METHOD

METHOD _copyToModel_SM_InnerRoom
  VAR_IN_OUT
    {attribute 'OPC.UA.DA' := '0'}
    model : M_SM_InnerRoom;
  END_VAR
                  model.actualStatus := THIS^.actualStatus;
model.setPoint := THIS^.setPoint;
model.avgTemp := THIS^.avgTemp;
model.avgPower := THIS^.avgPower;
model.totalPower := THIS^.totalPower;
model.ptpAvgTemp := THIS^.ptpAvgTemp;
model.ptpAllTemp := THIS^.ptpAllTemp;
model.stat := THIS^.stat;
THIS^.parts.tAbove._copyToModel_TempMeasurement( model := model.parts.tAbove );
THIS^.parts.tBelow._copyToModel_TempMeasurement( model := model.parts.tBelow );
THIS^.parts.tEast._copyToModel_TempMeasurement( model := model.parts.tEast );
THIS^.parts.tWest._copyToModel_TempMeasurement( model := model.parts.tWest );
THIS^.parts.htDucts._copyToModel_Heater( model := model.parts.htDucts );
THIS^.parts.ref._copyToModel_RefSensor( model := model.parts.ref );
THIS^.proc.initialize._copyToModel_Process( model := model.proc.initialize );
THIS^.proc.start._copyToModel_Process( model := model.proc.start );
THIS^.proc.stop._copyToModel_Process( model := model.proc.stop );
THIS^.proc.reset._copyToModel_Process( model := model.proc.reset );
THIS^.proc.clearPtp._copyToModel_Process( model := model.proc.clearPtp );
THIS^.proc.lock._copyToModel_Process( model := model.proc.lock );
THIS^.proc.unlock._copyToModel_Process( model := model.proc.unlock );

                
END_METHOD
END_FUNCTION_BLOCK

FUNCTION_BLOCK SM_Vessel
  VAR_INPUT
    {attribute 'OPC.UA.DA' := '1'}
    {attribute 'OPC.UA.DA.Access' := '1'}
    tStatBottomOk AT %I* : BOOL;  (* State of the thermostat switch at the vessel bottom *)
    {attribute 'OPC.UA.DA' := '1'}
    {attribute 'OPC.UA.DA.Access' := '1'}
    tStatLidOk AT %I* : BOOL;  (* State of the thermostat switch at the lid top *)
  END_VAR
  VAR_OUTPUT
    {attribute 'OPC.UA.DA' := '1'}
    {attribute 'OPC.UA.DA.Access' := '1'}
    actualStatus : STRING(50);  (* Current status description *)
    {attribute 'OPC.UA.DA' := '1'}
    {attribute 'OPC.UA.DA.Access' := '1'}
    setPoint : LREAL;  (* The ramped setpoint used by the pid *)
    {attribute 'OPC.UA.DA' := '1'}
    {attribute 'OPC.UA.DA.Access' := '1'}
    avgTemp : LREAL;  (* Average temperature of the vessel in kelvin *)
    {attribute 'OPC.UA.DA' := '1'}
    {attribute 'OPC.UA.DA.Access' := '1'}
    avgPower : LREAL;  (* Average power of the heaters in percentage *)
    {attribute 'OPC.UA.DA' := '1'}
    {attribute 'OPC.UA.DA.Access' := '1'}
    totalPower : LREAL;  (* Total power of all heaters in watt *)
    {attribute 'OPC.UA.DA' := '1'}
    {attribute 'OPC.UA.DA.Access' := '1'}
    ptpAvgTemp : ARRAY[1..5] OF LREAL;  (* ptp values of the average temperature of the vessel" *)
    {attribute 'OPC.UA.DA' := '1'}
    {attribute 'OPC.UA.DA.Access' := '1'}
    ptpAllTemp : ARRAY[1..5] OF LREAL;  (* ptp values of all temp measurements in the vessel" *)
    {attribute 'OPC.UA.DA' := '1'}
    {attribute 'OPC.UA.DA.Access' := '1'}
    tStatBottomPwr AT %Q* : BOOL;  (* Thermostat switch vessel bottom power *)
    {attribute 'OPC.UA.DA' := '1'}
    {attribute 'OPC.UA.DA.Access' := '1'}
    tStatLidPwr AT %Q* : BOOL;  (* Thermostat switch lid top power *)
    {attribute 'OPC.UA.DA' := '1'}
    stat : VesselStatuses;  (* Statuses of the state machine *)
    {attribute 'OPC.UA.DA' := '1'}
    parts : VesselParts;  (* Parts of the state machine *)
    {attribute 'OPC.UA.DA' := '1'}
    proc : VesselProcesses;  (* Processes of the state machine *)
  END_VAR
  VAR_IN_OUT
    {attribute 'OPC.UA.DA' := '0'}
    config_ref : VesselConfig;  (* Active configuration of the vessel *)
    {attribute 'OPC.UA.DA' := '0'}
    sharedConfig_ref : ThermoSharedConfig;  (* Shared config for the thermo system *)
    {attribute 'OPC.UA.DA' := '0'}
    activity_ref : ActivityStatus;  (* Shared activity status *)
    {attribute 'OPC.UA.DA' := '0'}
    services_ref : Services;  (* Shared services *)
    {attribute 'OPC.UA.DA' := '0'}
    operator_ref : OperatorStatus;  (* Shared operator status *)
  END_VAR

            parts.tLegNE(
    config_ref := config_ref.tLegNE,
    sharedConfig_ref := config_ref.shared.sensors);
parts.tLegNW(
    config_ref := config_ref.tLegNW,
    sharedConfig_ref := config_ref.shared.sensors);
parts.tLegSE(
    config_ref := config_ref.tLegSE,
    sharedConfig_ref := config_ref.shared.sensors);
parts.tLegSW(
    config_ref := config_ref.tLegSW,
    sharedConfig_ref := config_ref.shared.sensors);
parts.tLegTopNE(
    config_ref := config_ref.tLegTopNE,
    sharedConfig_ref := config_ref.shared.sensors);
parts.tLegTopNW(
    config_ref := config_ref.tLegTopNW,
    sharedConfig_ref := config_ref.shared.sensors);
parts.tLegTopSE(
    config_ref := config_ref.tLegTopSE,
    sharedConfig_ref := config_ref.shared.sensors);
parts.tLegTopSW(
    config_ref := config_ref.tLegTopSW,
    sharedConfig_ref := config_ref.shared.sensors);
parts.tBotNE(
    config_ref := config_ref.tBotNE,
    sharedConfig_ref := config_ref.shared.sensors);
parts.tBotNW(
    config_ref := config_ref.tBotNW,
    sharedConfig_ref := config_ref.shared.sensors);
parts.tBotSE(
    config_ref := config_ref.tBotSE,
    sharedConfig_ref := config_ref.shared.sensors);
parts.tBotSW(
    config_ref := config_ref.tBotSW,
    sharedConfig_ref := config_ref.shared.sensors);
parts.tCenter(
    config_ref := config_ref.tCenter,
    sharedConfig_ref := config_ref.shared.sensors);
parts.tCenterTH10K(
    config_ref := config_ref.tCenterTH10K,
    sharedConfig_ref := config_ref.shared.sensors);
parts.tSideN(
    config_ref := config_ref.tSideN,
    sharedConfig_ref := config_ref.shared.sensors);
parts.tSideS(
    config_ref := config_ref.tSideS,
    sharedConfig_ref := config_ref.shared.sensors);
parts.tSideE(
    config_ref := config_ref.tSideE,
    sharedConfig_ref := config_ref.shared.sensors);
parts.tSideW(
    config_ref := config_ref.tSideW,
    sharedConfig_ref := config_ref.shared.sensors);
parts.tLidN(
    config_ref := config_ref.tLidN,
    sharedConfig_ref := config_ref.shared.sensors);
parts.tLidS(
    config_ref := config_ref.tLidS,
    sharedConfig_ref := config_ref.shared.sensors);
parts.htLegNE(
    config_ref := config_ref.htLegNE,
    sharedConfig_ref := config_ref.shared.heaters,
    operator_ref := operator_ref);
parts.htLegNW(
    config_ref := config_ref.htLegNW,
    sharedConfig_ref := config_ref.shared.heaters,
    operator_ref := operator_ref);
parts.htLegSE(
    config_ref := config_ref.htLegSE,
    sharedConfig_ref := config_ref.shared.heaters,
    operator_ref := operator_ref);
parts.htLegSW(
    config_ref := config_ref.htLegSW,
    sharedConfig_ref := config_ref.shared.heaters,
    operator_ref := operator_ref);
parts.htLegTopNE(
    config_ref := config_ref.htLegTopNE,
    sharedConfig_ref := config_ref.shared.heaters,
    operator_ref := operator_ref);
parts.htLegTopNW(
    config_ref := config_ref.htLegTopNW,
    sharedConfig_ref := config_ref.shared.heaters,
    operator_ref := operator_ref);
parts.htLegTopSE(
    config_ref := config_ref.htLegTopSE,
    sharedConfig_ref := config_ref.shared.heaters,
    operator_ref := operator_ref);
parts.htLegTopSW(
    config_ref := config_ref.htLegTopSW,
    sharedConfig_ref := config_ref.shared.heaters,
    operator_ref := operator_ref);
parts.htBotNE(
    config_ref := config_ref.htBotNE,
    sharedConfig_ref := config_ref.shared.heaters,
    operator_ref := operator_ref);
parts.htBotNW(
    config_ref := config_ref.htBotNW,
    sharedConfig_ref := config_ref.shared.heaters,
    operator_ref := operator_ref);
parts.htBotSE(
    config_ref := config_ref.htBotSE,
    sharedConfig_ref := config_ref.shared.heaters,
    operator_ref := operator_ref);
parts.htBotSW(
    config_ref := config_ref.htBotSW,
    sharedConfig_ref := config_ref.shared.heaters,
    operator_ref := operator_ref);
parts.htSideN(
    config_ref := config_ref.htSideN,
    sharedConfig_ref := config_ref.shared.heaters,
    operator_ref := operator_ref);
parts.htSideS(
    config_ref := config_ref.htSideS,
    sharedConfig_ref := config_ref.shared.heaters,
    operator_ref := operator_ref);
parts.htSideE(
    config_ref := config_ref.htSideE,
    sharedConfig_ref := config_ref.shared.heaters,
    operator_ref := operator_ref);
parts.htSideW(
    config_ref := config_ref.htSideW,
    sharedConfig_ref := config_ref.shared.heaters,
    operator_ref := operator_ref);
parts.htLidN(
    config_ref := config_ref.htLidN,
    sharedConfig_ref := config_ref.shared.heaters,
    operator_ref := operator_ref);
parts.htLidS(
    config_ref := config_ref.htLidS,
    sharedConfig_ref := config_ref.shared.heaters,
    operator_ref := operator_ref);
parts.ref();
stat.enabled := F_EnabledStatus(
    superState := TRUE,
    isEnabled := config_ref.enabled);
stat.busy := F_BusyStatus(
    superState := TRUE,
    isBusy := (stat.control = TempControlStatus.warming_up) OR (stat.init = InitializationStatus.initializing));
proc.initialize( isEnabled := NOT((stat.init = InitializationStatus.locked) OR (stat.enabled = EnabledStatus.disabled)) );
proc.start( isEnabled := (stat.control = TempControlStatus.idle) AND ((stat.init = InitializationStatus.initialized) AND (stat.enabled = EnabledStatus.enabled)) );
proc.stop( isEnabled := (NOT(stat.control = TempControlStatus.idle)) AND (stat.init = InitializationStatus.initialized) );
proc.reset( isEnabled := TRUE );
proc.clearPtp( isEnabled := (operator_ref = OperatorStatus.tech) AND (stat.init = InitializationStatus.initialized) );
proc.lock( isEnabled := (operator_ref = OperatorStatus.tech) AND (NOT(stat.init = InitializationStatus.locked)) );
proc.unlock( isEnabled := (operator_ref = OperatorStatus.tech) AND (stat.init = InitializationStatus.locked) );

          

METHOD _copyFromModel_SM_Vessel
  VAR_IN_OUT
    {attribute 'OPC.UA.DA' := '0'}
    model : M_SM_Vessel;
  END_VAR
                  THIS^.parts.tLegNE._copyFromModel_TempMeasurement( model := model.parts.tLegNE );
THIS^.parts.tLegNW._copyFromModel_TempMeasurement( model := model.parts.tLegNW );
THIS^.parts.tLegSE._copyFromModel_TempMeasurement( model := model.parts.tLegSE );
THIS^.parts.tLegSW._copyFromModel_TempMeasurement( model := model.parts.tLegSW );
THIS^.parts.tLegTopNE._copyFromModel_TempMeasurement( model := model.parts.tLegTopNE );
THIS^.parts.tLegTopNW._copyFromModel_TempMeasurement( model := model.parts.tLegTopNW );
THIS^.parts.tLegTopSE._copyFromModel_TempMeasurement( model := model.parts.tLegTopSE );
THIS^.parts.tLegTopSW._copyFromModel_TempMeasurement( model := model.parts.tLegTopSW );
THIS^.parts.tBotNE._copyFromModel_TempMeasurement( model := model.parts.tBotNE );
THIS^.parts.tBotNW._copyFromModel_TempMeasurement( model := model.parts.tBotNW );
THIS^.parts.tBotSE._copyFromModel_TempMeasurement( model := model.parts.tBotSE );
THIS^.parts.tBotSW._copyFromModel_TempMeasurement( model := model.parts.tBotSW );
THIS^.parts.tCenter._copyFromModel_TempMeasurement( model := model.parts.tCenter );
THIS^.parts.tCenterTH10K._copyFromModel_TempMeasurement( model := model.parts.tCenterTH10K );
THIS^.parts.tSideN._copyFromModel_TempMeasurement( model := model.parts.tSideN );
THIS^.parts.tSideS._copyFromModel_TempMeasurement( model := model.parts.tSideS );
THIS^.parts.tSideE._copyFromModel_TempMeasurement( model := model.parts.tSideE );
THIS^.parts.tSideW._copyFromModel_TempMeasurement( model := model.parts.tSideW );
THIS^.parts.tLidN._copyFromModel_TempMeasurement( model := model.parts.tLidN );
THIS^.parts.tLidS._copyFromModel_TempMeasurement( model := model.parts.tLidS );
THIS^.parts.htLegNE._copyFromModel_Heater( model := model.parts.htLegNE );
THIS^.parts.htLegNW._copyFromModel_Heater( model := model.parts.htLegNW );
THIS^.parts.htLegSE._copyFromModel_Heater( model := model.parts.htLegSE );
THIS^.parts.htLegSW._copyFromModel_Heater( model := model.parts.htLegSW );
THIS^.parts.htLegTopNE._copyFromModel_Heater( model := model.parts.htLegTopNE );
THIS^.parts.htLegTopNW._copyFromModel_Heater( model := model.parts.htLegTopNW );
THIS^.parts.htLegTopSE._copyFromModel_Heater( model := model.parts.htLegTopSE );
THIS^.parts.htLegTopSW._copyFromModel_Heater( model := model.parts.htLegTopSW );
THIS^.parts.htBotNE._copyFromModel_Heater( model := model.parts.htBotNE );
THIS^.parts.htBotNW._copyFromModel_Heater( model := model.parts.htBotNW );
THIS^.parts.htBotSE._copyFromModel_Heater( model := model.parts.htBotSE );
THIS^.parts.htBotSW._copyFromModel_Heater( model := model.parts.htBotSW );
THIS^.parts.htSideN._copyFromModel_Heater( model := model.parts.htSideN );
THIS^.parts.htSideS._copyFromModel_Heater( model := model.parts.htSideS );
THIS^.parts.htSideE._copyFromModel_Heater( model := model.parts.htSideE );
THIS^.parts.htSideW._copyFromModel_Heater( model := model.parts.htSideW );
THIS^.parts.htLidN._copyFromModel_Heater( model := model.parts.htLidN );
THIS^.parts.htLidS._copyFromModel_Heater( model := model.parts.htLidS );
THIS^.parts.ref._copyFromModel_RefSensor( model := model.parts.ref );
THIS^.proc.initialize._copyFromModel_Process( model := model.proc.initialize );
THIS^.proc.start._copyFromModel_Process( model := model.proc.start );
THIS^.proc.stop._copyFromModel_Process( model := model.proc.stop );
THIS^.proc.reset._copyFromModel_Process( model := model.proc.reset );
THIS^.proc.clearPtp._copyFromModel_Process( model := model.proc.clearPtp );
THIS^.proc.lock._copyFromModel_Process( model := model.proc.lock );
THIS^.proc.unlock._copyFromModel_Process( model := model.proc.unlock );

                
END_METHOD

METHOD _copyToModel_SM_Vessel
  VAR_IN_OUT
    {attribute 'OPC.UA.DA' := '0'}
    model : M_SM_Vessel;
  END_VAR
                  model.tStatBottomOk := THIS^.tStatBottomOk;
model.tStatLidOk := THIS^.tStatLidOk;
model.actualStatus := THIS^.actualStatus;
model.setPoint := THIS^.setPoint;
model.avgTemp := THIS^.avgTemp;
model.avgPower := THIS^.avgPower;
model.totalPower := THIS^.totalPower;
model.ptpAvgTemp := THIS^.ptpAvgTemp;
model.ptpAllTemp := THIS^.ptpAllTemp;
model.tStatBottomPwr := THIS^.tStatBottomPwr;
model.tStatLidPwr := THIS^.tStatLidPwr;
model.stat := THIS^.stat;
THIS^.parts.tLegNE._copyToModel_TempMeasurement( model := model.parts.tLegNE );
THIS^.parts.tLegNW._copyToModel_TempMeasurement( model := model.parts.tLegNW );
THIS^.parts.tLegSE._copyToModel_TempMeasurement( model := model.parts.tLegSE );
THIS^.parts.tLegSW._copyToModel_TempMeasurement( model := model.parts.tLegSW );
THIS^.parts.tLegTopNE._copyToModel_TempMeasurement( model := model.parts.tLegTopNE );
THIS^.parts.tLegTopNW._copyToModel_TempMeasurement( model := model.parts.tLegTopNW );
THIS^.parts.tLegTopSE._copyToModel_TempMeasurement( model := model.parts.tLegTopSE );
THIS^.parts.tLegTopSW._copyToModel_TempMeasurement( model := model.parts.tLegTopSW );
THIS^.parts.tBotNE._copyToModel_TempMeasurement( model := model.parts.tBotNE );
THIS^.parts.tBotNW._copyToModel_TempMeasurement( model := model.parts.tBotNW );
THIS^.parts.tBotSE._copyToModel_TempMeasurement( model := model.parts.tBotSE );
THIS^.parts.tBotSW._copyToModel_TempMeasurement( model := model.parts.tBotSW );
THIS^.parts.tCenter._copyToModel_TempMeasurement( model := model.parts.tCenter );
THIS^.parts.tCenterTH10K._copyToModel_TempMeasurement( model := model.parts.tCenterTH10K );
THIS^.parts.tSideN._copyToModel_TempMeasurement( model := model.parts.tSideN );
THIS^.parts.tSideS._copyToModel_TempMeasurement( model := model.parts.tSideS );
THIS^.parts.tSideE._copyToModel_TempMeasurement( model := model.parts.tSideE );
THIS^.parts.tSideW._copyToModel_TempMeasurement( model := model.parts.tSideW );
THIS^.parts.tLidN._copyToModel_TempMeasurement( model := model.parts.tLidN );
THIS^.parts.tLidS._copyToModel_TempMeasurement( model := model.parts.tLidS );
THIS^.parts.htLegNE._copyToModel_Heater( model := model.parts.htLegNE );
THIS^.parts.htLegNW._copyToModel_Heater( model := model.parts.htLegNW );
THIS^.parts.htLegSE._copyToModel_Heater( model := model.parts.htLegSE );
THIS^.parts.htLegSW._copyToModel_Heater( model := model.parts.htLegSW );
THIS^.parts.htLegTopNE._copyToModel_Heater( model := model.parts.htLegTopNE );
THIS^.parts.htLegTopNW._copyToModel_Heater( model := model.parts.htLegTopNW );
THIS^.parts.htLegTopSE._copyToModel_Heater( model := model.parts.htLegTopSE );
THIS^.parts.htLegTopSW._copyToModel_Heater( model := model.parts.htLegTopSW );
THIS^.parts.htBotNE._copyToModel_Heater( model := model.parts.htBotNE );
THIS^.parts.htBotNW._copyToModel_Heater( model := model.parts.htBotNW );
THIS^.parts.htBotSE._copyToModel_Heater( model := model.parts.htBotSE );
THIS^.parts.htBotSW._copyToModel_Heater( model := model.parts.htBotSW );
THIS^.parts.htSideN._copyToModel_Heater( model := model.parts.htSideN );
THIS^.parts.htSideS._copyToModel_Heater( model := model.parts.htSideS );
THIS^.parts.htSideE._copyToModel_Heater( model := model.parts.htSideE );
THIS^.parts.htSideW._copyToModel_Heater( model := model.parts.htSideW );
THIS^.parts.htLidN._copyToModel_Heater( model := model.parts.htLidN );
THIS^.parts.htLidS._copyToModel_Heater( model := model.parts.htLidS );
THIS^.parts.ref._copyToModel_RefSensor( model := model.parts.ref );
THIS^.proc.initialize._copyToModel_Process( model := model.proc.initialize );
THIS^.proc.start._copyToModel_Process( model := model.proc.start );
THIS^.proc.stop._copyToModel_Process( model := model.proc.stop );
THIS^.proc.reset._copyToModel_Process( model := model.proc.reset );
THIS^.proc.clearPtp._copyToModel_Process( model := model.proc.clearPtp );
THIS^.proc.lock._copyToModel_Process( model := model.proc.lock );
THIS^.proc.unlock._copyToModel_Process( model := model.proc.unlock );

                
END_METHOD
END_FUNCTION_BLOCK

FUNCTION_BLOCK SM_Shield
  VAR_OUTPUT
    {attribute 'OPC.UA.DA' := '1'}
    {attribute 'OPC.UA.DA.Access' := '1'}
    actualStatus : STRING(50);  (* Current status description *)
    {attribute 'OPC.UA.DA' := '1'}
    {attribute 'OPC.UA.DA.Access' := '1'}
    setPoint : LREAL;  (* The ramped setpoint used by the pid *)
    {attribute 'OPC.UA.DA' := '1'}
    {attribute 'OPC.UA.DA.Access' := '1'}
    avgTemp : LREAL;  (* Average temperature of the vessel in kelvin *)
    {attribute 'OPC.UA.DA' := '1'}
    {attribute 'OPC.UA.DA.Access' := '1'}
    avgPower : LREAL;  (* Average power of the heaters in percentage *)
    {attribute 'OPC.UA.DA' := '1'}
    {attribute 'OPC.UA.DA.Access' := '1'}
    totalPower : LREAL;  (* Total power of all heaters in watt *)
    {attribute 'OPC.UA.DA' := '1'}
    {attribute 'OPC.UA.DA.Access' := '1'}
    ptpAvgTemp : ARRAY[1..5] OF LREAL;  (* ptp values of the average temperature of the vessel" *)
    {attribute 'OPC.UA.DA' := '1'}
    {attribute 'OPC.UA.DA.Access' := '1'}
    ptpAllTemp : ARRAY[1..5] OF LREAL;  (* ptp values of all temp measurements in the vessel" *)
    {attribute 'OPC.UA.DA' := '1'}
    stat : ShieldStatuses;  (* Statuses of the state machine *)
    {attribute 'OPC.UA.DA' := '1'}
    parts : ShieldParts;  (* Parts of the state machine *)
    {attribute 'OPC.UA.DA' := '1'}
    proc : ShieldProcesses;  (* Processes of the state machine *)
  END_VAR
  VAR_IN_OUT
    {attribute 'OPC.UA.DA' := '0'}
    config_ref : ShieldConfig;  (* Active configuration of the shield *)
    {attribute 'OPC.UA.DA' := '0'}
    sharedConfig_ref : ThermoSharedConfig;  (* Shared config for the thermo system *)
    {attribute 'OPC.UA.DA' := '0'}
    activity_ref : ActivityStatus;  (* Shared activity status *)
    {attribute 'OPC.UA.DA' := '0'}
    services_ref : Services;  (* Shared services *)
    {attribute 'OPC.UA.DA' := '0'}
    operator_ref : OperatorStatus;  (* Shared operator status *)
  END_VAR

            parts.tTopNE(
    config_ref := config_ref.tTopNE,
    sharedConfig_ref := config_ref.shared.sensors);
parts.tTopNW(
    config_ref := config_ref.tTopNW,
    sharedConfig_ref := config_ref.shared.sensors);
parts.tTopSE(
    config_ref := config_ref.tTopSE,
    sharedConfig_ref := config_ref.shared.sensors);
parts.tTopSW(
    config_ref := config_ref.tTopSW,
    sharedConfig_ref := config_ref.shared.sensors);
parts.tSideN(
    config_ref := config_ref.tSideN,
    sharedConfig_ref := config_ref.shared.sensors);
parts.tSideS(
    config_ref := config_ref.tSideS,
    sharedConfig_ref := config_ref.shared.sensors);
parts.tSideNE(
    config_ref := config_ref.tSideNE,
    sharedConfig_ref := config_ref.shared.sensors);
parts.tSideSE(
    config_ref := config_ref.tSideSE,
    sharedConfig_ref := config_ref.shared.sensors);
parts.tSideNW(
    config_ref := config_ref.tSideNW,
    sharedConfig_ref := config_ref.shared.sensors);
parts.tSideSW(
    config_ref := config_ref.tSideSW,
    sharedConfig_ref := config_ref.shared.sensors);
parts.tBotNE(
    config_ref := config_ref.tBotNE,
    sharedConfig_ref := config_ref.shared.sensors);
parts.tBotNW(
    config_ref := config_ref.tBotNW,
    sharedConfig_ref := config_ref.shared.sensors);
parts.tBotS(
    config_ref := config_ref.tBotS,
    sharedConfig_ref := config_ref.shared.sensors);
parts.tCentre(
    config_ref := config_ref.tCentre,
    sharedConfig_ref := config_ref.shared.sensors);
parts.tCentreTh10k(
    config_ref := config_ref.tCentreTh10k,
    sharedConfig_ref := config_ref.shared.sensors);
parts.htTopNE(
    config_ref := config_ref.htTopNE,
    sharedConfig_ref := config_ref.shared.heaters,
    operator_ref := operator_ref);
parts.htTopNW(
    config_ref := config_ref.htTopNW,
    sharedConfig_ref := config_ref.shared.heaters,
    operator_ref := operator_ref);
parts.htTopSE(
    config_ref := config_ref.htTopSE,
    sharedConfig_ref := config_ref.shared.heaters,
    operator_ref := operator_ref);
parts.htTopSW(
    config_ref := config_ref.htTopSW,
    sharedConfig_ref := config_ref.shared.heaters,
    operator_ref := operator_ref);
parts.htSideN(
    config_ref := config_ref.htSideN,
    sharedConfig_ref := config_ref.shared.heaters,
    operator_ref := operator_ref);
parts.htSideS(
    config_ref := config_ref.htSideS,
    sharedConfig_ref := config_ref.shared.heaters,
    operator_ref := operator_ref);
parts.htSideNE(
    config_ref := config_ref.htSideNE,
    sharedConfig_ref := config_ref.shared.heaters,
    operator_ref := operator_ref);
parts.htSideSE(
    config_ref := config_ref.htSideSE,
    sharedConfig_ref := config_ref.shared.heaters,
    operator_ref := operator_ref);
parts.htSideNW(
    config_ref := config_ref.htSideNW,
    sharedConfig_ref := config_ref.shared.heaters,
    operator_ref := operator_ref);
parts.htSideSW(
    config_ref := config_ref.htSideSW,
    sharedConfig_ref := config_ref.shared.heaters,
    operator_ref := operator_ref);
parts.htBotNE(
    config_ref := config_ref.htBotNE,
    sharedConfig_ref := config_ref.shared.heaters,
    operator_ref := operator_ref);
parts.htBotNW(
    config_ref := config_ref.htBotNW,
    sharedConfig_ref := config_ref.shared.heaters,
    operator_ref := operator_ref);
parts.htBotS(
    config_ref := config_ref.htBotS,
    sharedConfig_ref := config_ref.shared.heaters,
    operator_ref := operator_ref);
parts.htCentre(
    config_ref := config_ref.htCentre,
    sharedConfig_ref := config_ref.shared.heaters,
    operator_ref := operator_ref);
parts.ref();
stat.enabled := F_EnabledStatus(
    superState := TRUE,
    isEnabled := config_ref.enabled);
stat.busy := F_BusyStatus(
    superState := TRUE,
    isBusy := (stat.control = TempControlStatus.warming_up) OR (stat.init = InitializationStatus.initializing));
proc.initialize( isEnabled := NOT((stat.init = InitializationStatus.locked) OR (stat.enabled = EnabledStatus.disabled)) );
proc.start( isEnabled := (stat.control = TempControlStatus.idle) AND ((stat.init = InitializationStatus.initialized) AND (stat.enabled = EnabledStatus.enabled)) );
proc.stop( isEnabled := (NOT(stat.control = TempControlStatus.idle)) AND (stat.init = InitializationStatus.initialized) );
proc.reset( isEnabled := TRUE );
proc.clearPtp( isEnabled := (operator_ref = OperatorStatus.tech) AND (stat.init = InitializationStatus.initialized) );
proc.lock( isEnabled := (operator_ref = OperatorStatus.tech) AND (NOT(stat.init = InitializationStatus.locked)) );
proc.unlock( isEnabled := (operator_ref = OperatorStatus.tech) AND (stat.init = InitializationStatus.locked) );

          

METHOD _copyFromModel_SM_Shield
  VAR_IN_OUT
    {attribute 'OPC.UA.DA' := '0'}
    model : M_SM_Shield;
  END_VAR
                  THIS^.parts.tTopNE._copyFromModel_TempMeasurement( model := model.parts.tTopNE );
THIS^.parts.tTopNW._copyFromModel_TempMeasurement( model := model.parts.tTopNW );
THIS^.parts.tTopSE._copyFromModel_TempMeasurement( model := model.parts.tTopSE );
THIS^.parts.tTopSW._copyFromModel_TempMeasurement( model := model.parts.tTopSW );
THIS^.parts.tSideN._copyFromModel_TempMeasurement( model := model.parts.tSideN );
THIS^.parts.tSideS._copyFromModel_TempMeasurement( model := model.parts.tSideS );
THIS^.parts.tSideNE._copyFromModel_TempMeasurement( model := model.parts.tSideNE );
THIS^.parts.tSideSE._copyFromModel_TempMeasurement( model := model.parts.tSideSE );
THIS^.parts.tSideNW._copyFromModel_TempMeasurement( model := model.parts.tSideNW );
THIS^.parts.tSideSW._copyFromModel_TempMeasurement( model := model.parts.tSideSW );
THIS^.parts.tBotNE._copyFromModel_TempMeasurement( model := model.parts.tBotNE );
THIS^.parts.tBotNW._copyFromModel_TempMeasurement( model := model.parts.tBotNW );
THIS^.parts.tBotS._copyFromModel_TempMeasurement( model := model.parts.tBotS );
THIS^.parts.tCentre._copyFromModel_TempMeasurement( model := model.parts.tCentre );
THIS^.parts.tCentreTh10k._copyFromModel_TempMeasurement( model := model.parts.tCentreTh10k );
THIS^.parts.htTopNE._copyFromModel_Heater( model := model.parts.htTopNE );
THIS^.parts.htTopNW._copyFromModel_Heater( model := model.parts.htTopNW );
THIS^.parts.htTopSE._copyFromModel_Heater( model := model.parts.htTopSE );
THIS^.parts.htTopSW._copyFromModel_Heater( model := model.parts.htTopSW );
THIS^.parts.htSideN._copyFromModel_Heater( model := model.parts.htSideN );
THIS^.parts.htSideS._copyFromModel_Heater( model := model.parts.htSideS );
THIS^.parts.htSideNE._copyFromModel_Heater( model := model.parts.htSideNE );
THIS^.parts.htSideSE._copyFromModel_Heater( model := model.parts.htSideSE );
THIS^.parts.htSideNW._copyFromModel_Heater( model := model.parts.htSideNW );
THIS^.parts.htSideSW._copyFromModel_Heater( model := model.parts.htSideSW );
THIS^.parts.htBotNE._copyFromModel_Heater( model := model.parts.htBotNE );
THIS^.parts.htBotNW._copyFromModel_Heater( model := model.parts.htBotNW );
THIS^.parts.htBotS._copyFromModel_Heater( model := model.parts.htBotS );
THIS^.parts.htCentre._copyFromModel_Heater( model := model.parts.htCentre );
THIS^.parts.ref._copyFromModel_RefSensor( model := model.parts.ref );
THIS^.proc.initialize._copyFromModel_Process( model := model.proc.initialize );
THIS^.proc.start._copyFromModel_Process( model := model.proc.start );
THIS^.proc.stop._copyFromModel_Process( model := model.proc.stop );
THIS^.proc.reset._copyFromModel_Process( model := model.proc.reset );
THIS^.proc.clearPtp._copyFromModel_Process( model := model.proc.clearPtp );
THIS^.proc.lock._copyFromModel_Process( model := model.proc.lock );
THIS^.proc.unlock._copyFromModel_Process( model := model.proc.unlock );

                
END_METHOD

METHOD _copyToModel_SM_Shield
  VAR_IN_OUT
    {attribute 'OPC.UA.DA' := '0'}
    model : M_SM_Shield;
  END_VAR
                  model.actualStatus := THIS^.actualStatus;
model.setPoint := THIS^.setPoint;
model.avgTemp := THIS^.avgTemp;
model.avgPower := THIS^.avgPower;
model.totalPower := THIS^.totalPower;
model.ptpAvgTemp := THIS^.ptpAvgTemp;
model.ptpAllTemp := THIS^.ptpAllTemp;
model.stat := THIS^.stat;
THIS^.parts.tTopNE._copyToModel_TempMeasurement( model := model.parts.tTopNE );
THIS^.parts.tTopNW._copyToModel_TempMeasurement( model := model.parts.tTopNW );
THIS^.parts.tTopSE._copyToModel_TempMeasurement( model := model.parts.tTopSE );
THIS^.parts.tTopSW._copyToModel_TempMeasurement( model := model.parts.tTopSW );
THIS^.parts.tSideN._copyToModel_TempMeasurement( model := model.parts.tSideN );
THIS^.parts.tSideS._copyToModel_TempMeasurement( model := model.parts.tSideS );
THIS^.parts.tSideNE._copyToModel_TempMeasurement( model := model.parts.tSideNE );
THIS^.parts.tSideSE._copyToModel_TempMeasurement( model := model.parts.tSideSE );
THIS^.parts.tSideNW._copyToModel_TempMeasurement( model := model.parts.tSideNW );
THIS^.parts.tSideSW._copyToModel_TempMeasurement( model := model.parts.tSideSW );
THIS^.parts.tBotNE._copyToModel_TempMeasurement( model := model.parts.tBotNE );
THIS^.parts.tBotNW._copyToModel_TempMeasurement( model := model.parts.tBotNW );
THIS^.parts.tBotS._copyToModel_TempMeasurement( model := model.parts.tBotS );
THIS^.parts.tCentre._copyToModel_TempMeasurement( model := model.parts.tCentre );
THIS^.parts.tCentreTh10k._copyToModel_TempMeasurement( model := model.parts.tCentreTh10k );
THIS^.parts.htTopNE._copyToModel_Heater( model := model.parts.htTopNE );
THIS^.parts.htTopNW._copyToModel_Heater( model := model.parts.htTopNW );
THIS^.parts.htTopSE._copyToModel_Heater( model := model.parts.htTopSE );
THIS^.parts.htTopSW._copyToModel_Heater( model := model.parts.htTopSW );
THIS^.parts.htSideN._copyToModel_Heater( model := model.parts.htSideN );
THIS^.parts.htSideS._copyToModel_Heater( model := model.parts.htSideS );
THIS^.parts.htSideNE._copyToModel_Heater( model := model.parts.htSideNE );
THIS^.parts.htSideSE._copyToModel_Heater( model := model.parts.htSideSE );
THIS^.parts.htSideNW._copyToModel_Heater( model := model.parts.htSideNW );
THIS^.parts.htSideSW._copyToModel_Heater( model := model.parts.htSideSW );
THIS^.parts.htBotNE._copyToModel_Heater( model := model.parts.htBotNE );
THIS^.parts.htBotNW._copyToModel_Heater( model := model.parts.htBotNW );
THIS^.parts.htBotS._copyToModel_Heater( model := model.parts.htBotS );
THIS^.parts.htCentre._copyToModel_Heater( model := model.parts.htCentre );
THIS^.parts.ref._copyToModel_RefSensor( model := model.parts.ref );
THIS^.proc.initialize._copyToModel_Process( model := model.proc.initialize );
THIS^.proc.start._copyToModel_Process( model := model.proc.start );
THIS^.proc.stop._copyToModel_Process( model := model.proc.stop );
THIS^.proc.reset._copyToModel_Process( model := model.proc.reset );
THIS^.proc.clearPtp._copyToModel_Process( model := model.proc.clearPtp );
THIS^.proc.lock._copyToModel_Process( model := model.proc.lock );
THIS^.proc.unlock._copyToModel_Process( model := model.proc.unlock );

                
END_METHOD
END_FUNCTION_BLOCK

FUNCTION_BLOCK SM_Bench
  VAR_OUTPUT
    {attribute 'OPC.UA.DA' := '1'}
    {attribute 'OPC.UA.DA.Access' := '1'}
    actualStatus : STRING(50);  (* Current status description *)
    {attribute 'OPC.UA.DA' := '1'}
    stat : BenchStatuses;  (* Statuses of the state machine *)
    {attribute 'OPC.UA.DA' := '1'}
    parts : BenchParts;  (* Parts of the state machine *)
    {attribute 'OPC.UA.DA' := '1'}
    proc : BenchProcesses;  (* Processes of the state machine *)
  END_VAR
  VAR_IN_OUT
    {attribute 'OPC.UA.DA' := '0'}
    config_ref : BenchConfig;  (* Active configuration of the bench *)
    {attribute 'OPC.UA.DA' := '0'}
    sharedConfig_ref : ThermoSharedConfig;  (* Shared config for the thermo system *)
    {attribute 'OPC.UA.DA' := '0'}
    activity_ref : ActivityStatus;  (* Shared activity status *)
    {attribute 'OPC.UA.DA' := '0'}
    services_ref : Services;  (* Shared services *)
    {attribute 'OPC.UA.DA' := '0'}
    operator_ref : OperatorStatus;  (* Shared operator status *)
  END_VAR

            parts.tCentre(
    config_ref := config_ref.tCentre,
    sharedConfig_ref := config_ref.shared.sensors);
parts.tCentreTH10k(
    config_ref := config_ref.tCentreTH10k,
    sharedConfig_ref := config_ref.shared.sensors);
parts.tCollBench(
    config_ref := config_ref.tCollBench,
    sharedConfig_ref := config_ref.shared.sensors);
parts.tEchelleCryo(
    config_ref := config_ref.tEchelleCryo,
    sharedConfig_ref := config_ref.shared.sensors);
parts.tCamCryo(
    config_ref := config_ref.tCamCryo,
    sharedConfig_ref := config_ref.shared.sensors);
parts.tColl(
    config_ref := config_ref.tColl,
    sharedConfig_ref := config_ref.shared.sensors);
parts.tPrism(
    config_ref := config_ref.tPrism,
    sharedConfig_ref := config_ref.shared.sensors);
parts.tEchelle(
    config_ref := config_ref.tEchelle,
    sharedConfig_ref := config_ref.shared.sensors);
parts.tCam(
    config_ref := config_ref.tCam,
    sharedConfig_ref := config_ref.shared.sensors);
parts.tInOptics(
    config_ref := config_ref.tInOptics,
    sharedConfig_ref := config_ref.shared.sensors);
parts.htCollBench(
    config_ref := config_ref.htCollBench,
    sharedConfig_ref := config_ref.shared.heaters,
    operator_ref := operator_ref);
parts.htEchelleCryo(
    config_ref := config_ref.htEchelleCryo,
    sharedConfig_ref := config_ref.shared.heaters,
    operator_ref := operator_ref);
parts.htCamCryo(
    config_ref := config_ref.htCamCryo,
    sharedConfig_ref := config_ref.shared.heaters,
    operator_ref := operator_ref);
parts.htEchellePrism(
    config_ref := config_ref.htEchellePrism,
    sharedConfig_ref := config_ref.shared.heaters,
    operator_ref := operator_ref);
parts.ref();
stat.enabled := F_EnabledStatus(
    superState := TRUE,
    isEnabled := config_ref.enabled);
stat.busy := F_BusyStatus(
    superState := TRUE,
    isBusy := (stat.control = TempControlStatus.warming_up) OR (stat.init = InitializationStatus.initializing));
proc.initialize();
proc.start();
proc.stop();
proc.reset();
proc.clearPtp();
proc.lock();
proc.unlock();

          

METHOD _copyFromModel_SM_Bench
  VAR_IN_OUT
    {attribute 'OPC.UA.DA' := '0'}
    model : M_SM_Bench;
  END_VAR
                  THIS^.parts.tCentre._copyFromModel_TempMeasurement( model := model.parts.tCentre );
THIS^.parts.tCentreTH10k._copyFromModel_TempMeasurement( model := model.parts.tCentreTH10k );
THIS^.parts.tCollBench._copyFromModel_TempMeasurement( model := model.parts.tCollBench );
THIS^.parts.tEchelleCryo._copyFromModel_TempMeasurement( model := model.parts.tEchelleCryo );
THIS^.parts.tCamCryo._copyFromModel_TempMeasurement( model := model.parts.tCamCryo );
THIS^.parts.tColl._copyFromModel_TempMeasurement( model := model.parts.tColl );
THIS^.parts.tPrism._copyFromModel_TempMeasurement( model := model.parts.tPrism );
THIS^.parts.tEchelle._copyFromModel_TempMeasurement( model := model.parts.tEchelle );
THIS^.parts.tCam._copyFromModel_TempMeasurement( model := model.parts.tCam );
THIS^.parts.tInOptics._copyFromModel_TempMeasurement( model := model.parts.tInOptics );
THIS^.parts.htCollBench._copyFromModel_Heater( model := model.parts.htCollBench );
THIS^.parts.htEchelleCryo._copyFromModel_Heater( model := model.parts.htEchelleCryo );
THIS^.parts.htCamCryo._copyFromModel_Heater( model := model.parts.htCamCryo );
THIS^.parts.htEchellePrism._copyFromModel_Heater( model := model.parts.htEchellePrism );
THIS^.parts.ref._copyFromModel_RefSensor( model := model.parts.ref );
THIS^.proc.initialize._copyFromModel_Process( model := model.proc.initialize );
THIS^.proc.start._copyFromModel_Process( model := model.proc.start );
THIS^.proc.stop._copyFromModel_Process( model := model.proc.stop );
THIS^.proc.reset._copyFromModel_Process( model := model.proc.reset );
THIS^.proc.clearPtp._copyFromModel_Process( model := model.proc.clearPtp );
THIS^.proc.lock._copyFromModel_Process( model := model.proc.lock );
THIS^.proc.unlock._copyFromModel_Process( model := model.proc.unlock );

                
END_METHOD

METHOD _copyToModel_SM_Bench
  VAR_IN_OUT
    {attribute 'OPC.UA.DA' := '0'}
    model : M_SM_Bench;
  END_VAR
                  model.actualStatus := THIS^.actualStatus;
model.stat := THIS^.stat;
THIS^.parts.tCentre._copyToModel_TempMeasurement( model := model.parts.tCentre );
THIS^.parts.tCentreTH10k._copyToModel_TempMeasurement( model := model.parts.tCentreTH10k );
THIS^.parts.tCollBench._copyToModel_TempMeasurement( model := model.parts.tCollBench );
THIS^.parts.tEchelleCryo._copyToModel_TempMeasurement( model := model.parts.tEchelleCryo );
THIS^.parts.tCamCryo._copyToModel_TempMeasurement( model := model.parts.tCamCryo );
THIS^.parts.tColl._copyToModel_TempMeasurement( model := model.parts.tColl );
THIS^.parts.tPrism._copyToModel_TempMeasurement( model := model.parts.tPrism );
THIS^.parts.tEchelle._copyToModel_TempMeasurement( model := model.parts.tEchelle );
THIS^.parts.tCam._copyToModel_TempMeasurement( model := model.parts.tCam );
THIS^.parts.tInOptics._copyToModel_TempMeasurement( model := model.parts.tInOptics );
THIS^.parts.htCollBench._copyToModel_Heater( model := model.parts.htCollBench );
THIS^.parts.htEchelleCryo._copyToModel_Heater( model := model.parts.htEchelleCryo );
THIS^.parts.htCamCryo._copyToModel_Heater( model := model.parts.htCamCryo );
THIS^.parts.htEchellePrism._copyToModel_Heater( model := model.parts.htEchellePrism );
THIS^.parts.ref._copyToModel_RefSensor( model := model.parts.ref );
THIS^.proc.initialize._copyToModel_Process( model := model.proc.initialize );
THIS^.proc.start._copyToModel_Process( model := model.proc.start );
THIS^.proc.stop._copyToModel_Process( model := model.proc.stop );
THIS^.proc.reset._copyToModel_Process( model := model.proc.reset );
THIS^.proc.clearPtp._copyToModel_Process( model := model.proc.clearPtp );
THIS^.proc.lock._copyToModel_Process( model := model.proc.lock );
THIS^.proc.unlock._copyToModel_Process( model := model.proc.unlock );

                
END_METHOD
END_FUNCTION_BLOCK

FUNCTION_BLOCK SM_Cryo
  VAR_INPUT
    {attribute 'OPC.UA.DA' := '1'}
    {attribute 'OPC.UA.DA.Access' := '1'}
    tStatCryoRearOk AT %I* : BOOL;  (* State of the thermostat switch at the cryo rear *)
  END_VAR
  VAR_OUTPUT
    {attribute 'OPC.UA.DA' := '1'}
    {attribute 'OPC.UA.DA.Access' := '1'}
    actualStatus : STRING(50);  (* Current status description *)
    {attribute 'OPC.UA.DA' := '1'}
    {attribute 'OPC.UA.DA.Access' := '1'}
    tStatCryoRearPwr AT %Q* : BOOL;  (* Thermostat switch cryo rear power *)
    {attribute 'OPC.UA.DA' := '1'}
    stat : CryoStatuses;  (* Statuses of the state machine *)
    {attribute 'OPC.UA.DA' := '1'}
    parts : CryoParts;  (* Parts of the state machine *)
    {attribute 'OPC.UA.DA' := '1'}
    proc : CryoProcesses;  (* Processes of the state machine *)
  END_VAR
  VAR_IN_OUT
    {attribute 'OPC.UA.DA' := '0'}
    config_ref : CryoConfig;  (* Active configuration of the bench *)
    {attribute 'OPC.UA.DA' := '0'}
    sharedConfig_ref : ThermoSharedConfig;  (* Shared config for the thermo system *)
    {attribute 'OPC.UA.DA' := '0'}
    activity_ref : ActivityStatus;  (* Shared activity status *)
    {attribute 'OPC.UA.DA' := '0'}
    services_ref : Services;  (* Shared services *)
    {attribute 'OPC.UA.DA' := '0'}
    operator_ref : OperatorStatus;  (* Shared operator status *)
  END_VAR

            parts.tRearOut(
    config_ref := config_ref.tRearOut,
    sharedConfig_ref := config_ref.shared.sensors);
parts.tRearIn(
    config_ref := config_ref.tRearIn,
    sharedConfig_ref := config_ref.shared.sensors);
parts.tFront(
    config_ref := config_ref.tFront,
    sharedConfig_ref := config_ref.shared.sensors);
parts.htRearOut(
    config_ref := config_ref.htRearOut,
    sharedConfig_ref := config_ref.shared.heaters,
    operator_ref := operator_ref);
parts.htRearIn(
    config_ref := config_ref.htRearIn,
    sharedConfig_ref := config_ref.shared.heaters,
    operator_ref := operator_ref);
parts.htRearFront(
    config_ref := config_ref.htRearFront,
    sharedConfig_ref := config_ref.shared.heaters,
    operator_ref := operator_ref);
parts.ref();
stat.enabled := F_EnabledStatus(
    superState := TRUE,
    isEnabled := config_ref.enabled);
stat.busy := F_BusyStatus(
    superState := TRUE,
    isBusy := (stat.control = TempControlStatus.warming_up) OR (stat.init = InitializationStatus.initializing));
proc.initialize();
proc.start();
proc.stop();
proc.reset();
proc.clearPtp();
proc.lock();
proc.unlock();

          

METHOD _copyFromModel_SM_Cryo
  VAR_IN_OUT
    {attribute 'OPC.UA.DA' := '0'}
    model : M_SM_Cryo;
  END_VAR
                  THIS^.parts.tRearOut._copyFromModel_TempMeasurement( model := model.parts.tRearOut );
THIS^.parts.tRearIn._copyFromModel_TempMeasurement( model := model.parts.tRearIn );
THIS^.parts.tFront._copyFromModel_TempMeasurement( model := model.parts.tFront );
THIS^.parts.htRearOut._copyFromModel_Heater( model := model.parts.htRearOut );
THIS^.parts.htRearIn._copyFromModel_Heater( model := model.parts.htRearIn );
THIS^.parts.htRearFront._copyFromModel_Heater( model := model.parts.htRearFront );
THIS^.parts.ref._copyFromModel_RefSensor( model := model.parts.ref );
THIS^.proc.initialize._copyFromModel_Process( model := model.proc.initialize );
THIS^.proc.start._copyFromModel_Process( model := model.proc.start );
THIS^.proc.stop._copyFromModel_Process( model := model.proc.stop );
THIS^.proc.reset._copyFromModel_Process( model := model.proc.reset );
THIS^.proc.clearPtp._copyFromModel_Process( model := model.proc.clearPtp );
THIS^.proc.lock._copyFromModel_Process( model := model.proc.lock );
THIS^.proc.unlock._copyFromModel_Process( model := model.proc.unlock );

                
END_METHOD

METHOD _copyToModel_SM_Cryo
  VAR_IN_OUT
    {attribute 'OPC.UA.DA' := '0'}
    model : M_SM_Cryo;
  END_VAR
                  model.tStatCryoRearOk := THIS^.tStatCryoRearOk;
model.actualStatus := THIS^.actualStatus;
model.tStatCryoRearPwr := THIS^.tStatCryoRearPwr;
model.stat := THIS^.stat;
THIS^.parts.tRearOut._copyToModel_TempMeasurement( model := model.parts.tRearOut );
THIS^.parts.tRearIn._copyToModel_TempMeasurement( model := model.parts.tRearIn );
THIS^.parts.tFront._copyToModel_TempMeasurement( model := model.parts.tFront );
THIS^.parts.htRearOut._copyToModel_Heater( model := model.parts.htRearOut );
THIS^.parts.htRearIn._copyToModel_Heater( model := model.parts.htRearIn );
THIS^.parts.htRearFront._copyToModel_Heater( model := model.parts.htRearFront );
THIS^.parts.ref._copyToModel_RefSensor( model := model.parts.ref );
THIS^.proc.initialize._copyToModel_Process( model := model.proc.initialize );
THIS^.proc.start._copyToModel_Process( model := model.proc.start );
THIS^.proc.stop._copyToModel_Process( model := model.proc.stop );
THIS^.proc.reset._copyToModel_Process( model := model.proc.reset );
THIS^.proc.clearPtp._copyToModel_Process( model := model.proc.clearPtp );
THIS^.proc.lock._copyToModel_Process( model := model.proc.lock );
THIS^.proc.unlock._copyToModel_Process( model := model.proc.unlock );

                
END_METHOD
END_FUNCTION_BLOCK

FUNCTION_BLOCK SM_Thermo
  VAR_OUTPUT
    {attribute 'OPC.UA.DA' := '1'}
    {attribute 'OPC.UA.DA.Access' := '1'}
    actualStatus : STRING(50);  (* Current status description *)
    {attribute 'OPC.UA.DA' := '1'}
    stat : ThermoStatuses;  (* Statuses of the state machine *)
    {attribute 'OPC.UA.DA' := '1'}
    parts : ThermoParts;  (* Parts of the state machine *)
    {attribute 'OPC.UA.DA' := '1'}
    proc : ThermoProcesses;  (* Processes of the state machine *)
  END_VAR
  VAR_IN_OUT
    {attribute 'OPC.UA.DA' := '0'}
    config_ref : ThermoConfig;  (* active configuration of the thermo control system *)
    {attribute 'OPC.UA.DA' := '0'}
    activity_ref : ActivityStatus;  (* Shared activity status *)
    {attribute 'OPC.UA.DA' := '0'}
    services_ref : Services;  (* Shared services *)
    {attribute 'OPC.UA.DA' := '0'}
    operator_ref : OperatorStatus;  (* Shared operator status *)
  END_VAR

            parts.outerRoom(
    activity_ref := activity_ref,
    services_ref := services_ref,
    operator_ref := operator_ref,
    config_ref := config_ref.outerRoom,
    sharedConfig_ref := config_ref.shared);
parts.innerRoom(
    activity_ref := activity_ref,
    services_ref := services_ref,
    operator_ref := operator_ref,
    config_ref := config_ref.innerRoom,
    sharedConfig_ref := config_ref.shared);
parts.vessel(
    activity_ref := activity_ref,
    services_ref := services_ref,
    operator_ref := operator_ref,
    config_ref := config_ref.vessel,
    sharedConfig_ref := config_ref.shared);
parts.shield(
    activity_ref := activity_ref,
    services_ref := services_ref,
    operator_ref := operator_ref,
    config_ref := config_ref.shield,
    sharedConfig_ref := config_ref.shared);
parts.bench(
    activity_ref := activity_ref,
    services_ref := services_ref,
    operator_ref := operator_ref,
    config_ref := config_ref.bench,
    sharedConfig_ref := config_ref.shared);
parts.cryo(
    activity_ref := activity_ref,
    services_ref := services_ref,
    operator_ref := operator_ref,
    config_ref := config_ref.cryo,
    sharedConfig_ref := config_ref.shared);
stat.enabled := F_EnabledStatus(
    superState := TRUE,
    isEnabled := config_ref.enabled);
stat.busy := F_BusyStatus(
    superState := NOT(stat.init = InitializationStatus.shutdown),
    isBusy := ((parts.outerRoom.stat.busy = BusyStatus.busy) OR ((parts.innerRoom.stat.busy = BusyStatus.busy) OR ((parts.vessel.stat.busy = BusyStatus.busy) OR ((parts.shield.stat.busy = BusyStatus.busy) OR ((parts.bench.stat.busy = BusyStatus.busy) OR (parts.cryo.stat.busy = BusyStatus.busy)))))) OR (stat.init = InitializationStatus.initializing));
stat.control := F_TempControlStatus(
    superState := stat.init = InitializationStatus.initialized,
    isWarmingUp := (parts.outerRoom.stat.control = TempControlStatus.warming_up) OR ((parts.innerRoom.stat.control = TempControlStatus.warming_up) OR ((parts.vessel.stat.control = TempControlStatus.warming_up) OR ((parts.shield.stat.control = TempControlStatus.warming_up) OR ((parts.bench.stat.control = TempControlStatus.warming_up) OR (parts.cryo.stat.control = TempControlStatus.warming_up))))),
    isActive := (parts.outerRoom.stat.control = TempControlStatus.active) OR ((parts.innerRoom.stat.control = TempControlStatus.active) OR ((parts.vessel.stat.control = TempControlStatus.active) OR ((parts.shield.stat.control = TempControlStatus.active) OR ((parts.bench.stat.control = TempControlStatus.active) OR (parts.cryo.stat.control = TempControlStatus.active))))));
proc.initialize( isEnabled := NOT((stat.init = InitializationStatus.locked) OR (stat.enabled = EnabledStatus.disabled)) );
proc.start( isEnabled := (stat.control = TempControlStatus.idle) AND ((stat.init = InitializationStatus.initialized) AND (stat.enabled = EnabledStatus.enabled)) );
proc.stop( isEnabled := (NOT(stat.control = TempControlStatus.idle)) AND (stat.init = InitializationStatus.initialized) );
proc.clearPtp( isEnabled := (operator_ref = OperatorStatus.tech) AND (stat.init = InitializationStatus.initialized) );
proc.reset( isEnabled := TRUE );
proc.lock( isEnabled := (operator_ref = OperatorStatus.tech) AND (NOT(stat.init = InitializationStatus.locked)) );
proc.unlock( isEnabled := (operator_ref = OperatorStatus.tech) AND (stat.init = InitializationStatus.locked) );

          

METHOD _copyFromModel_SM_Thermo
  VAR_IN_OUT
    {attribute 'OPC.UA.DA' := '0'}
    model : M_SM_Thermo;
  END_VAR
                  THIS^.parts.outerRoom._copyFromModel_OuterRoom( model := model.parts.outerRoom );
THIS^.parts.innerRoom._copyFromModel_InnerRoom( model := model.parts.innerRoom );
THIS^.parts.vessel._copyFromModel_Vessel( model := model.parts.vessel );
THIS^.parts.shield._copyFromModel_Shield( model := model.parts.shield );
THIS^.parts.bench._copyFromModel_Bench( model := model.parts.bench );
THIS^.parts.cryo._copyFromModel_Cryo( model := model.parts.cryo );
THIS^.proc.initialize._copyFromModel_Process( model := model.proc.initialize );
THIS^.proc.start._copyFromModel_Process( model := model.proc.start );
THIS^.proc.stop._copyFromModel_Process( model := model.proc.stop );
THIS^.proc.clearPtp._copyFromModel_Process( model := model.proc.clearPtp );
THIS^.proc.reset._copyFromModel_Process( model := model.proc.reset );
THIS^.proc.lock._copyFromModel_Process( model := model.proc.lock );
THIS^.proc.unlock._copyFromModel_Process( model := model.proc.unlock );

                
END_METHOD

METHOD _copyToModel_SM_Thermo
  VAR_IN_OUT
    {attribute 'OPC.UA.DA' := '0'}
    model : M_SM_Thermo;
  END_VAR
                  model.actualStatus := THIS^.actualStatus;
model.stat := THIS^.stat;
THIS^.parts.outerRoom._copyToModel_OuterRoom( model := model.parts.outerRoom );
THIS^.parts.innerRoom._copyToModel_InnerRoom( model := model.parts.innerRoom );
THIS^.parts.vessel._copyToModel_Vessel( model := model.parts.vessel );
THIS^.parts.shield._copyToModel_Shield( model := model.parts.shield );
THIS^.parts.bench._copyToModel_Bench( model := model.parts.bench );
THIS^.parts.cryo._copyToModel_Cryo( model := model.parts.cryo );
THIS^.proc.initialize._copyToModel_Process( model := model.proc.initialize );
THIS^.proc.start._copyToModel_Process( model := model.proc.start );
THIS^.proc.stop._copyToModel_Process( model := model.proc.stop );
THIS^.proc.clearPtp._copyToModel_Process( model := model.proc.clearPtp );
THIS^.proc.reset._copyToModel_Process( model := model.proc.reset );
THIS^.proc.lock._copyToModel_Process( model := model.proc.lock );
THIS^.proc.unlock._copyToModel_Process( model := model.proc.unlock );

                
END_METHOD
END_FUNCTION_BLOCK

FUNCTION_BLOCK SM_Vac
  VAR_OUTPUT
    {attribute 'OPC.UA.DA' := '1'}
    {attribute 'OPC.UA.DA.Access' := '1'}
    actualStatus : STRING(50);  (* Current status description *)
    {attribute 'OPC.UA.DA' := '1'}
    stat : VacStatuses;  (* Statuses of the state machine *)
    {attribute 'OPC.UA.DA' := '1'}
    proc : VacProcesses;  (* Processes of the state machine *)
  END_VAR
  VAR_IN_OUT
    {attribute 'OPC.UA.DA' := '0'}
    config_ref : VacConfig;  (* active configuration of the thermo control system *)
    {attribute 'OPC.UA.DA' := '0'}
    activity_ref : ActivityStatus;  (* Shared activity status *)
    {attribute 'OPC.UA.DA' := '0'}
    services_ref : Services;  (* Shared services *)
    {attribute 'OPC.UA.DA' := '0'}
    operator_ref : OperatorStatus;  (* Shared operator status *)
  END_VAR

            stat.enabled := F_EnabledStatus(
    superState := TRUE,
    isEnabled := config_ref.enabled);
proc.initialize( isEnabled := NOT((stat.init = InitializationStatus.locked) OR (stat.enabled = EnabledStatus.disabled)) );
proc.reset( isEnabled := TRUE );
proc.lock( isEnabled := (operator_ref = OperatorStatus.tech) AND (NOT(stat.init = InitializationStatus.locked)) );
proc.unlock( isEnabled := (operator_ref = OperatorStatus.tech) AND (stat.init = InitializationStatus.locked) );

          

METHOD _copyFromModel_SM_Vac
  VAR_IN_OUT
    {attribute 'OPC.UA.DA' := '0'}
    model : M_SM_Vac;
  END_VAR
                  THIS^.proc.initialize._copyFromModel_Process( model := model.proc.initialize );
THIS^.proc.reset._copyFromModel_Process( model := model.proc.reset );
THIS^.proc.lock._copyFromModel_Process( model := model.proc.lock );
THIS^.proc.unlock._copyFromModel_Process( model := model.proc.unlock );

                
END_METHOD

METHOD _copyToModel_SM_Vac
  VAR_IN_OUT
    {attribute 'OPC.UA.DA' := '0'}
    model : M_SM_Vac;
  END_VAR
                  model.actualStatus := THIS^.actualStatus;
model.stat := THIS^.stat;
THIS^.proc.initialize._copyToModel_Process( model := model.proc.initialize );
THIS^.proc.reset._copyToModel_Process( model := model.proc.reset );
THIS^.proc.lock._copyToModel_Process( model := model.proc.lock );
THIS^.proc.unlock._copyToModel_Process( model := model.proc.unlock );

                
END_METHOD
END_FUNCTION_BLOCK

FUNCTION_BLOCK SM_ThermoVac
  VAR_INPUT
    {attribute 'OPC.UA.DA' := '1'}
    {attribute 'OPC.UA.DA.Access' := '3'}
    editableConfig : ThermoVacConfig;  (* Editable configuration of the thermo vac system *)
  END_VAR
  VAR_OUTPUT
    {attribute 'OPC.UA.DA' := '1'}
    {attribute 'OPC.UA.DA.Access' := '1'}
    actualStatus : STRING(50);  (* Current status description *)
    {attribute 'OPC.UA.DA' := '1'}
    {attribute 'OPC.UA.DA.Access' := '1'}
    config : ThermoVacConfig;  (* active configuration of the thermo vac system *)
    {attribute 'OPC.UA.DA' := '1'}
    stat : ThermoVacStatuses;  (* Statuses of the state machine *)
    {attribute 'OPC.UA.DA' := '1'}
    parts : ThermoVacParts;  (* Parts of the state machine *)
    {attribute 'OPC.UA.DA' := '1'}
    proc : ThermoVacProcesses;  (* Processes of the state machine *)
  END_VAR
  VAR_IN_OUT
    {attribute 'OPC.UA.DA' := '0'}
    activity_ref : ActivityStatus;  (* Shared activity status *)
    {attribute 'OPC.UA.DA' := '0'}
    services_ref : Services;  (* Shared services *)
    {attribute 'OPC.UA.DA' := '0'}
    operator_ref : OperatorStatus;  (* Shared operator status *)
  END_VAR

            parts.thermo(
    activity_ref := activity_ref,
    services_ref := services_ref,
    operator_ref := operator_ref,
    config_ref := config.thermo);
parts.vac(
    activity_ref := activity_ref,
    services_ref := services_ref,
    operator_ref := operator_ref,
    config_ref := config.vac);
parts.configManager( isEnabled := operator_ref = OperatorStatus.tech );
stat.busy := F_BusyStatus(
    superState := NOT(stat.init = InitializationStatus.shutdown),
    isBusy := ((parts.thermo.stat.busy = BusyStatus.busy) OR (parts.vac.stat.busy = BusyStatus.busy)) OR (stat.init = InitializationStatus.initializing));
proc.initialize( isEnabled := NOT(stat.init = InitializationStatus.locked) );
proc.reset( isEnabled := TRUE );
proc.lock( isEnabled := (operator_ref = OperatorStatus.tech) AND (NOT(stat.init = InitializationStatus.locked)) );
proc.unlock( isEnabled := (operator_ref = OperatorStatus.tech) AND (stat.init = InitializationStatus.locked) );

          

METHOD _copyFromModel_SM_ThermoVac
  VAR_IN_OUT
    {attribute 'OPC.UA.DA' := '0'}
    model : M_SM_ThermoVac;
  END_VAR
                  THIS^.editableConfig := model.editableConfig;
THIS^.parts.thermo._copyFromModel_Thermo( model := model.parts.thermo );
THIS^.parts.vac._copyFromModel_Vac( model := model.parts.vac );
THIS^.parts.configManager._copyFromModel_ConfigManager( model := model.parts.configManager );
THIS^.proc.initialize._copyFromModel_Process( model := model.proc.initialize );
THIS^.proc.reset._copyFromModel_Process( model := model.proc.reset );
THIS^.proc.lock._copyFromModel_Process( model := model.proc.lock );
THIS^.proc.unlock._copyFromModel_Process( model := model.proc.unlock );

                
END_METHOD

